(* IEC 61131-3 sources: SmartHomeNew/ (part 11) *)

(* ---- PRG_Config_Staged_Change_Monitor.st ---- *)
PROGRAM PRG_Config_Staged_Change_Monitor
// ==============================================================================
// CONFIG STAGED CHANGE MONITOR
// ==============================================================================
// Tracks generic staged config fields controlled by GVL_CONFIG_CONTROL. When any
// staged value changes, the staged config version is incremented so HMI validation
// cannot be reused for a different draft.
// ==============================================================================
VAR
    L_Initialized : BOOL;
    L_Changed : BOOL;

    L_Last_STG_Reputation_Learning_Rate : REAL;
    L_Last_STG_Reputation_Recovery_Decay : REAL;
    L_Last_STG_Min_Sensor_Confidence : REAL;
    L_Last_STG_Bad_Spike_Confidence : REAL;
    L_Last_STG_Default_Confidence : REAL;

    L_Last_STG_Night_Start_Hour : INT;
    L_Last_STG_Night_End_Hour : INT;
    L_Last_STG_VentBoost_Humidity_Threshold : REAL;

    L_Last_STG_Stabilization_Delay_MS : UDINT;

    L_Last_STG_PLC_Inactive_Close_Gas : BOOL;
    L_Last_STG_PLC_Inactive_Stop_Boiler : BOOL;
    L_Last_STG_PLC_Inactive_Block_Heating : BOOL;
    L_Last_STG_PLC_Inactive_Stop_Vent : BOOL;
    L_Last_STG_PLC_Inactive_Block_Water : BOOL;
END_VAR

L_Changed := FALSE;

IF NOT L_Initialized THEN
    L_Initialized := TRUE;
ELSE
    IF L_Last_STG_Reputation_Learning_Rate <> GVL_CONFIG_CONTROL.STG_Reputation_Learning_Rate THEN L_Changed := TRUE; END_IF;
    IF L_Last_STG_Reputation_Recovery_Decay <> GVL_CONFIG_CONTROL.STG_Reputation_Recovery_Decay THEN L_Changed := TRUE; END_IF;
    IF L_Last_STG_Min_Sensor_Confidence <> GVL_CONFIG_CONTROL.STG_Min_Sensor_Confidence THEN L_Changed := TRUE; END_IF;
    IF L_Last_STG_Bad_Spike_Confidence <> GVL_CONFIG_CONTROL.STG_Bad_Spike_Confidence THEN L_Changed := TRUE; END_IF;
    IF L_Last_STG_Default_Confidence <> GVL_CONFIG_CONTROL.STG_Default_Confidence THEN L_Changed := TRUE; END_IF;

    IF L_Last_STG_Night_Start_Hour <> GVL_CONFIG_CONTROL.STG_Night_Start_Hour THEN L_Changed := TRUE; END_IF;
    IF L_Last_STG_Night_End_Hour <> GVL_CONFIG_CONTROL.STG_Night_End_Hour THEN L_Changed := TRUE; END_IF;
    IF L_Last_STG_VentBoost_Humidity_Threshold <> GVL_CONFIG_CONTROL.STG_VentBoost_Humidity_Threshold THEN L_Changed := TRUE; END_IF;

    IF L_Last_STG_Stabilization_Delay_MS <> GVL_CONFIG_CONTROL.STG_Stabilization_Delay_MS THEN L_Changed := TRUE; END_IF;

    IF L_Last_STG_PLC_Inactive_Close_Gas <> GVL_CONFIG_CONTROL.STG_PLC_Inactive_Close_Gas THEN L_Changed := TRUE; END_IF;
    IF L_Last_STG_PLC_Inactive_Stop_Boiler <> GVL_CONFIG_CONTROL.STG_PLC_Inactive_Stop_Boiler THEN L_Changed := TRUE; END_IF;
    IF L_Last_STG_PLC_Inactive_Block_Heating <> GVL_CONFIG_CONTROL.STG_PLC_Inactive_Block_Heating THEN L_Changed := TRUE; END_IF;
    IF L_Last_STG_PLC_Inactive_Stop_Vent <> GVL_CONFIG_CONTROL.STG_PLC_Inactive_Stop_Vent THEN L_Changed := TRUE; END_IF;
    IF L_Last_STG_PLC_Inactive_Block_Water <> GVL_CONFIG_CONTROL.STG_PLC_Inactive_Block_Water THEN L_Changed := TRUE; END_IF;
END_IF;

IF L_Changed THEN
    GVL_CONFIG_CONTROL.G_Staged_Config_Version := GVL_CONFIG_CONTROL.G_Staged_Config_Version + 1;
    GVL_CONFIG_CONTROL.G_Staged_Last_Changed_MS := GVL_TIME_SERVICE.G_Now_MS;
END_IF;

L_Last_STG_Reputation_Learning_Rate := GVL_CONFIG_CONTROL.STG_Reputation_Learning_Rate;
L_Last_STG_Reputation_Recovery_Decay := GVL_CONFIG_CONTROL.STG_Reputation_Recovery_Decay;
L_Last_STG_Min_Sensor_Confidence := GVL_CONFIG_CONTROL.STG_Min_Sensor_Confidence;
L_Last_STG_Bad_Spike_Confidence := GVL_CONFIG_CONTROL.STG_Bad_Spike_Confidence;
L_Last_STG_Default_Confidence := GVL_CONFIG_CONTROL.STG_Default_Confidence;

L_Last_STG_Night_Start_Hour := GVL_CONFIG_CONTROL.STG_Night_Start_Hour;
L_Last_STG_Night_End_Hour := GVL_CONFIG_CONTROL.STG_Night_End_Hour;
L_Last_STG_VentBoost_Humidity_Threshold := GVL_CONFIG_CONTROL.STG_VentBoost_Humidity_Threshold;

L_Last_STG_Stabilization_Delay_MS := GVL_CONFIG_CONTROL.STG_Stabilization_Delay_MS;

L_Last_STG_PLC_Inactive_Close_Gas := GVL_CONFIG_CONTROL.STG_PLC_Inactive_Close_Gas;
L_Last_STG_PLC_Inactive_Stop_Boiler := GVL_CONFIG_CONTROL.STG_PLC_Inactive_Stop_Boiler;
L_Last_STG_PLC_Inactive_Block_Heating := GVL_CONFIG_CONTROL.STG_PLC_Inactive_Block_Heating;
L_Last_STG_PLC_Inactive_Stop_Vent := GVL_CONFIG_CONTROL.STG_PLC_Inactive_Stop_Vent;
L_Last_STG_PLC_Inactive_Block_Water := GVL_CONFIG_CONTROL.STG_PLC_Inactive_Block_Water;

// >>> BULK_SYNC_ANCHOR: PRG_Config_Staged_Change_Monitor <<<
END_PROGRAM

(* ---- PRG_Config_Validation.st ---- *)
PROGRAM PRG_Config_Validation
VAR
    fbConfigSimulation : FB_Config_Simulation;

    L_i : INT;
    L_Zone : INT;
    L_Sensor : INT;
    L_Manifold : INT;
    L_Map_Index : INT;
    L_Config_Error : BOOL;
END_VAR

// ======================================================
// CENTRAL CONFIGURATION VALIDATION
// ======================================================
// Diagnostic-only layer.
//
// This PRG may set validation/configuration status flags and text,
// but must not directly mutate aggregated diagnostics fields.
// Aggregated diagnostics ownership is centralized in:
//
//   FB_System_Health_Orchestrator
//
// This PRG also must not write command/shadow/output structures.
// ======================================================

L_Config_Error := FALSE;

// ======================================================
// ACTIVE SIZE CONFIGURATION
// ======================================================
IF (GVL_SYSTEM_SIZE_CONFIG.G_Active_Heating_Circuits < 1) OR
   (GVL_SYSTEM_SIZE_CONFIG.G_Active_Heating_Circuits > GVL_CONSTANTS.C_MAX_HEATING_CIRCUITS) THEN
    L_Config_Error := TRUE;
END_IF;

IF (GVL_SYSTEM_SIZE_CONFIG.G_Active_Water_Zones < 1) OR
   (GVL_SYSTEM_SIZE_CONFIG.G_Active_Water_Zones > GVL_CONSTANTS.C_MAX_WATER_ZONES) THEN
    L_Config_Error := TRUE;
END_IF;

IF (GVL_SYSTEM_SIZE_CONFIG.G_Active_Light_Zones < 1) OR
   (GVL_SYSTEM_SIZE_CONFIG.G_Active_Light_Zones > GVL_CONSTANTS.C_MAX_LIGHT_ZONES) THEN
    L_Config_Error := TRUE;
END_IF;

IF (GVL_SYSTEM_SIZE_CONFIG.G_Active_Blinds < 0) OR
   (GVL_SYSTEM_SIZE_CONFIG.G_Active_Blinds > GVL_CONSTANTS.C_MAX_BLINDS) THEN
    L_Config_Error := TRUE;
END_IF;

IF (GVL_SYSTEM_SIZE_CONFIG.G_Active_Sockets < 0) OR
   (GVL_SYSTEM_SIZE_CONFIG.G_Active_Sockets > GVL_CONSTANTS.C_MAX_SOCKETS) THEN
    L_Config_Error := TRUE;
END_IF;

// ======================================================
// HEATING CIRCUIT CONFIGURATION
// ======================================================
FOR L_i := 1 TO GVL_CONSTANTS.C_MAX_HEATING_CIRCUITS DO
    L_Zone := BYTE_TO_INT(GVL_CONFIG.G_HMI_FloorHeating_Configs[L_i].zone);
    L_Sensor := BYTE_TO_INT(GVL_CONFIG.G_HMI_FloorHeating_Configs[L_i].sensor_id);
    L_Manifold := BYTE_TO_INT(GVL_CONFIG.G_HMI_FloorHeating_Configs[L_i].manifold_id);

    IF (L_Zone < 1) OR (L_Zone > GVL_CONSTANTS.C_MAX_ZONES) THEN
        L_Config_Error := TRUE;
    END_IF;

    IF (L_Sensor < 1) OR (L_Sensor > GVL_CONSTANTS.C_MAX_ZONES) THEN
        L_Config_Error := TRUE;
    END_IF;

    IF (L_Manifold < 1) OR (L_Manifold > GVL_CONSTANTS.C_MAX_MANIFOLDS) THEN
        L_Config_Error := TRUE;
    END_IF;

    IF GVL_CONFIG.G_HMI_FloorHeating_Configs[L_i].min_temp > GVL_CONFIG.G_HMI_FloorHeating_Configs[L_i].max_temp THEN
        L_Config_Error := TRUE;
    END_IF;
END_FOR;

IF (GVL_CONFIG.G_Max_Active_Manifolds < 1) OR
   (GVL_CONFIG.G_Max_Active_Manifolds > GVL_CONSTANTS.C_MAX_MANIFOLDS) THEN
    L_Config_Error := TRUE;
END_IF;

IF GVL_CONFIG.G_Max_Thermal_Budget <= 0.0 THEN
    L_Config_Error := TRUE;
END_IF;

IF GVL_CONFIG.G_Policy_Min_Hold_MS < 10000 THEN
    L_Config_Error := TRUE;
END_IF;

// ======================================================
// ACCESS / TIMING CONFIGURATION
// ======================================================
IF (GVL_CONFIG.G_Access_Pulse_MS < 100) OR (GVL_CONFIG.G_Access_Pulse_MS > 5000) THEN
    L_Config_Error := TRUE;
END_IF;

// ======================================================
// MAP CONFIGURATION
// ======================================================
FOR L_i := 1 TO GVL_CONSTANTS.C_MAX_DOOR_SENSORS DO
    L_Map_Index := GVL_CONFIG.G_Door_Map[L_i];
    IF (L_Map_Index < 1) OR (L_Map_Index > GVL_CONSTANTS.C_MAX_SECURITY_SENSORS) THEN
        L_Config_Error := TRUE;
    END_IF;
END_FOR;

FOR L_i := 1 TO GVL_CONSTANTS.C_MAX_ZONES DO
    L_Map_Index := GVL_CONFIG.G_Window_Map[L_i];
    IF L_Map_Index <> 0 THEN
        IF (L_Map_Index < 1) OR (L_Map_Index > (GVL_CONSTANTS.C_MAX_SECURITY_SENSORS * 2)) THEN
            L_Config_Error := TRUE;
        END_IF;
    END_IF;
END_FOR;

FOR L_i := 1 TO GVL_CONSTANTS.C_MAX_HEATING_CIRCUITS DO
    IF (GVL_CONFIG.G_FloorTemp_Map[L_i] < 1) OR (GVL_CONFIG.G_FloorTemp_Map[L_i] > GVL_CONSTANTS.C_MAX_ZONES) THEN
        L_Config_Error := TRUE;
    END_IF;
END_FOR;

FOR L_i := 1 TO GVL_CONSTANTS.C_MAX_ZONES DO
    IF (GVL_CONFIG.G_RoomTemp_Map[L_i] < 1) OR (GVL_CONFIG.G_RoomTemp_Map[L_i] > GVL_CONSTANTS.C_MAX_ZONES) THEN
        L_Config_Error := TRUE;
    END_IF;
END_FOR;

// ======================================================
// HARDWARE SERVICE / RETRY CONFIGURATION
// ======================================================
IF GVL_CONFIG.G_Freeze_Hardware_Retry_Count < 0 THEN
    L_Config_Error := TRUE;
END_IF;

IF GVL_CONFIG.G_Freeze_Hardware_Retry_Delay_MS < 1000 THEN
    L_Config_Error := TRUE;
END_IF;

IF GVL_CONFIG.G_Pump_Exercise_Enabled THEN
    IF GVL_CONFIG.G_Pump_Exercise_Interval_MS < GVL_CONSTANTS.C_MS_IN_MINUTE THEN
        L_Config_Error := TRUE;
    END_IF;
    IF GVL_CONFIG.G_Pump_Exercise_Duration_MS < 1000 THEN
        L_Config_Error := TRUE;
    END_IF;
END_IF;

IF GVL_CONFIG.G_Water_Valve_Exercise_Enabled THEN
    IF GVL_CONFIG.G_Water_Valve_Exercise_Interval_MS < GVL_CONSTANTS.C_MS_IN_MINUTE THEN
        L_Config_Error := TRUE;
    END_IF;
    IF GVL_CONFIG.G_Water_Valve_Exercise_Duration_MS < 1000 THEN
        L_Config_Error := TRUE;
    END_IF;
END_IF;

IF GVL_CONFIG.G_Water_Valve_Close_Retry_Count < 0 THEN
    L_Config_Error := TRUE;
END_IF;

IF GVL_CONFIG.G_Water_Valve_Close_Retry_Delay_MS < 1000 THEN
    L_Config_Error := TRUE;
END_IF;

// ======================================================
// OPENTHERM / MODBUS RTU CONFIGURATION
// ======================================================
IF GVL_CONFIG.G_OpenTherm_Enabled THEN

    IF GVL_CONFIG.G_OpenTherm_Heartbeat_Timeout_MS < 1000 THEN
        L_Config_Error := TRUE;
    END_IF;

    IF GVL_CONFIG.G_OpenTherm_Command_Ack_Timeout_MS < 500 THEN
        L_Config_Error := TRUE;
    END_IF;

    IF GVL_CONFIG.G_Modbus_RTU_Baudrate < 1200 THEN
        L_Config_Error := TRUE;
    END_IF;

    IF (GVL_CONFIG.G_Modbus_RTU_Parity > 2) THEN
        L_Config_Error := TRUE;
    END_IF;

    IF (GVL_CONFIG.G_Modbus_RTU_Stop_Bits < 1) OR
       (GVL_CONFIG.G_Modbus_RTU_Stop_Bits > 2) THEN
        L_Config_Error := TRUE;
    END_IF;

    IF (GVL_CONFIG.G_Modbus_RTU_Data_Bits < 7) OR
       (GVL_CONFIG.G_Modbus_RTU_Data_Bits > 8) THEN
        L_Config_Error := TRUE;
    END_IF;

    IF GVL_CONFIG.G_Modbus_RTU_Slave_ID = 0 THEN
        L_Config_Error := TRUE;
    END_IF;

    IF GVL_CONFIG.G_Modbus_RTU_Poll_Interval_MS < 50 THEN
        L_Config_Error := TRUE;
    END_IF;

    IF GVL_CONFIG.G_Modbus_RTU_Request_Timeout_MS < 50 THEN
        L_Config_Error := TRUE;
    END_IF;

    IF GVL_CONFIG.G_Modbus_RTU_Retry_Count < 0 THEN
        L_Config_Error := TRUE;
    END_IF;

    FOR L_i := 1 TO GVL_CONSTANTS.C_MAX_BOILERS DO
        IF GVL_CONFIG.G_OpenTherm_Register_Map[L_i].Cmd_Enable_Offset = GVL_CONFIG.G_OpenTherm_Register_Map[L_i].Status_Word_Offset THEN
            L_Config_Error := TRUE;
        END_IF;

        IF GVL_CONFIG.G_OpenTherm_Register_Map[L_i].Cmd_Setpoint_x10_Offset = GVL_CONFIG.G_OpenTherm_Register_Map[L_i].Status_Word_Offset THEN
            L_Config_Error := TRUE;
        END_IF;
    END_FOR;
END_IF;

// ======================================================
// SENSOR COUNT SANITY
// ======================================================
IF GVL_CONSTANTS.C_MAX_METHANE_SENSORS < 2 THEN
    L_Config_Error := TRUE;
END_IF;

IF GVL_CONSTANTS.C_MAX_SMOKE_SENSORS < 6 THEN
    L_Config_Error := TRUE;
END_IF;

IF GVL_CONSTANTS.C_MAX_CO_SENSORS < 8 THEN
    L_Config_Error := TRUE;
END_IF;

IF GVL_CONSTANTS.C_MAX_FLOOD_SENSORS < 9 THEN
    L_Config_Error := TRUE;
END_IF;

// ======================================================
// CONFIG SIMULATION / COMMISSIONING VALIDATION
// ======================================================
fbConfigSimulation(
    VI_Enable := TRUE,
    VI_Request := GVL_CONFIG_SIMULATION.G_Simulation_Request,
    VI_Confirm := GVL_CONFIG_SIMULATION.G_Simulation_Confirm
);

IF fbConfigSimulation.VO_Executed AND NOT fbConfigSimulation.VO_Result_OK THEN
    L_Config_Error := TRUE;
END_IF;

// ======================================================
// STORE FLAGS
// ======================================================
GVL_CONFIG_VALIDATION.G_Config_Valid := NOT L_Config_Error;
GVL_CONFIG_VALIDATION.G_Config_Critical_Error := L_Config_Error;
GVL_CONFIG_VALIDATION.G_Config_Last_Update_MS := GVL_STATUS.G_System_Time_MS;

IF L_Config_Error THEN
    GVL_CONFIG_VALIDATION.G_Config_Active_Error_Text := 'CONFIG VALIDATION ERROR';
    GVL_STATUS.G_System_Mode_Text := 'CONFIG ERROR';
ELSE
    GVL_CONFIG_VALIDATION.G_Config_Active_Error_Text := '';
END_IF;

IF GVL_CONFIG_VALIDATION.G_Config_Active_Error_Text <> '' THEN
    GVL_CONFIG_VALIDATION.G_Config_Last_Error_Text := GVL_CONFIG_VALIDATION.G_Config_Active_Error_Text;
ELSIF GVL_CONFIG_VALIDATION.G_Config_Control_Error_Text <> '' THEN
    GVL_CONFIG_VALIDATION.G_Config_Last_Error_Text := GVL_CONFIG_VALIDATION.G_Config_Control_Error_Text;
ELSE
    GVL_CONFIG_VALIDATION.G_Config_Last_Error_Text := '';
END_IF;

END_PROGRAM

(* ---- PRG_Config_Versioning.st ---- *)
PROGRAM PRG_Config_Versioning
VAR
    L_i : INT;
    L_Config_Error : BOOL;
END_VAR

// Detect config error from validation layer.
// Calibration processor faults are surfaced through Sensor_Fault, so the
// configuration rollback snapshot must include calibration records too.
L_Config_Error := GVL_STATUS.G_Diagnostics.Sensor_Fault OR GVL_STATUS.G_Diagnostics.Subsystem_Degraded;

// --- Save snapshot when system is healthy ---
IF NOT L_Config_Error THEN
    FOR L_i := 1 TO GVL_CONSTANTS.C_MAX_HEATING_CIRCUITS DO
        GVL_CONFIG_BACKUP.G_Backup_FloorHeating_Configs[L_i] := GVL_CONFIG.G_HMI_FloorHeating_Configs[L_i];
    END_FOR;

    GVL_CONFIG_BACKUP.G_Backup_Max_Active_Manifolds := GVL_CONFIG.G_Max_Active_Manifolds;
    GVL_CONFIG_BACKUP.G_Backup_Max_Thermal_Budget := GVL_CONFIG.G_Max_Thermal_Budget;

    GVL_CONFIG_BACKUP.G_Backup_Calib_Outdoor_Temp := GVL_CONFIG.G_Calib_Outdoor_Temp;
    GVL_CONFIG_BACKUP.G_Backup_Calib_Ambient_Lux := GVL_CONFIG.G_Calib_Ambient_Lux;

    FOR L_i := 1 TO GVL_CONSTANTS.C_MAX_SUPPLY_TEMPS DO
        GVL_CONFIG_BACKUP.G_Backup_Calib_Supply_Temps[L_i] := GVL_CONFIG.G_Calib_Supply_Temps[L_i];
    END_FOR;

    FOR L_i := 1 TO GVL_CONSTANTS.C_MAX_ZONES DO
        GVL_CONFIG_BACKUP.G_Backup_Calib_Room_Temps[L_i] := GVL_CONFIG.G_Calib_Room_Temps[L_i];
        GVL_CONFIG_BACKUP.G_Backup_Calib_Floor_Temps[L_i] := GVL_CONFIG.G_Calib_Floor_Temps[L_i];
        GVL_CONFIG_BACKUP.G_Backup_Calib_CO2[L_i] := GVL_CONFIG.G_Calib_CO2[L_i];
        GVL_CONFIG_BACKUP.G_Backup_Calib_Humidity[L_i] := GVL_CONFIG.G_Calib_Humidity[L_i];
    END_FOR;

    FOR L_i := 1 TO GVL_CONSTANTS.C_MAX_MANIFOLDS DO
        GVL_CONFIG_BACKUP.G_Backup_Calib_Manifold_T_Supply[L_i] := GVL_CONFIG.G_Calib_Manifold_T_Supply[L_i];
        GVL_CONFIG_BACKUP.G_Backup_Calib_Manifold_T_Return[L_i] := GVL_CONFIG.G_Calib_Manifold_T_Return[L_i];
    END_FOR;

    FOR L_i := 1 TO GVL_CONSTANTS.C_MAX_METHANE_SENSORS DO
        GVL_CONFIG_BACKUP.G_Backup_Calib_Methane[L_i] := GVL_CONFIG.G_Calib_Methane[L_i];
    END_FOR;

    FOR L_i := 1 TO GVL_CONSTANTS.C_MAX_CO_SENSORS DO
        GVL_CONFIG_BACKUP.G_Backup_Calib_CO[L_i] := GVL_CONFIG.G_Calib_CO[L_i];
    END_FOR;

    GVL_CONFIG_BACKUP.G_Backup_Valid := TRUE;
END_IF;

// --- Rollback if config invalid ---
IF L_Config_Error THEN

    // Freeze system via command layer
    GVL_COMMAND_SHADOW.G_Heating_Block := TRUE;
    GVL_COMMAND_SHADOW.G_Boiler_Stop := TRUE;

    // Restore snapshot only if valid
    IF GVL_CONFIG_BACKUP.G_Backup_Valid THEN
        FOR L_i := 1 TO GVL_CONSTANTS.C_MAX_HEATING_CIRCUITS DO
            GVL_CONFIG.G_HMI_FloorHeating_Configs[L_i] := GVL_CONFIG_BACKUP.G_Backup_FloorHeating_Configs[L_i];
        END_FOR;

        GVL_CONFIG.G_Max_Active_Manifolds := GVL_CONFIG_BACKUP.G_Backup_Max_Active_Manifolds;
        GVL_CONFIG.G_Max_Thermal_Budget := GVL_CONFIG_BACKUP.G_Backup_Max_Thermal_Budget;

        GVL_CONFIG.G_Calib_Outdoor_Temp := GVL_CONFIG_BACKUP.G_Backup_Calib_Outdoor_Temp;
        GVL_CONFIG.G_Calib_Ambient_Lux := GVL_CONFIG_BACKUP.G_Backup_Calib_Ambient_Lux;

        FOR L_i := 1 TO GVL_CONSTANTS.C_MAX_SUPPLY_TEMPS DO
            GVL_CONFIG.G_Calib_Supply_Temps[L_i] := GVL_CONFIG_BACKUP.G_Backup_Calib_Supply_Temps[L_i];
        END_FOR;

        FOR L_i := 1 TO GVL_CONSTANTS.C_MAX_ZONES DO
            GVL_CONFIG.G_Calib_Room_Temps[L_i] := GVL_CONFIG_BACKUP.G_Backup_Calib_Room_Temps[L_i];
            GVL_CONFIG.G_Calib_Floor_Temps[L_i] := GVL_CONFIG_BACKUP.G_Backup_Calib_Floor_Temps[L_i];
            GVL_CONFIG.G_Calib_CO2[L_i] := GVL_CONFIG_BACKUP.G_Backup_Calib_CO2[L_i];
            GVL_CONFIG.G_Calib_Humidity[L_i] := GVL_CONFIG_BACKUP.G_Backup_Calib_Humidity[L_i];
        END_FOR;

        FOR L_i := 1 TO GVL_CONSTANTS.C_MAX_MANIFOLDS DO
            GVL_CONFIG.G_Calib_Manifold_T_Supply[L_i] := GVL_CONFIG_BACKUP.G_Backup_Calib_Manifold_T_Supply[L_i];
            GVL_CONFIG.G_Calib_Manifold_T_Return[L_i] := GVL_CONFIG_BACKUP.G_Backup_Calib_Manifold_T_Return[L_i];
        END_FOR;

        FOR L_i := 1 TO GVL_CONSTANTS.C_MAX_METHANE_SENSORS DO
            GVL_CONFIG.G_Calib_Methane[L_i] := GVL_CONFIG_BACKUP.G_Backup_Calib_Methane[L_i];
        END_FOR;

        FOR L_i := 1 TO GVL_CONSTANTS.C_MAX_CO_SENSORS DO
            GVL_CONFIG.G_Calib_CO[L_i] := GVL_CONFIG_BACKUP.G_Backup_Calib_CO[L_i];
        END_FOR;

        GVL_STATUS.G_System_Mode_Text := 'CONFIG ROLLBACK';
    ELSE
        GVL_STATUS.G_System_Mode_Text := 'CONFIG INVALID - NO BACKUP';
    END_IF;
END_IF;

END_PROGRAM
// >>> BULK_SYNC_ANCHOR: PRG_Config_Versioning <<<

(* ---- PRG_Convergence_Governor.st ---- *)
PROGRAM PRG_Convergence_Governor
VAR
    L_Now_MS : UDINT;
    L_Healthy : BOOL := TRUE;
    L_Error_Code : UDINT := 0;
    L_Error_Text : STRING(160) := '';
END_VAR

L_Now_MS := GVL_STATUS.G_System_Time_MS;
L_Healthy := TRUE;
L_Error_Code := 0;
L_Error_Text := '';

GVL_CONVERGENCE.Convergence_Runtime_Barrier_OK :=
    GVL_RUNTIME_EPOCH.Runtime_Runtime_Barrier_OK
    AND GVL_RUNTIME_EPOCH.Runtime_IO_Publication_Allowed;

GVL_CONVERGENCE.Convergence_Runtime_Snapshot_OK :=
    GVL_RUNTIME_SNAPSHOT.Snapshot_Frozen
    AND GVL_RUNTIME_SNAPSHOT.Snapshot_Publication_Allowed
    AND GVL_RUNTIME_SNAPSHOT.Snapshot_Copy_Valid
    AND GVL_RUNTIME_SNAPSHOT.Snapshot_Isolation_Valid
    AND GVL_RUNTIME_SNAPSHOT.Snapshot_Runtime_Authority_Valid
    AND NOT GVL_RUNTIME_SNAPSHOT.Snapshot_Mutation_Detected;

GVL_CONVERGENCE.Convergence_Distributed_Snapshot_OK :=
    GVL_DISTRIBUTED_SNAPSHOT.Distributed_Publication_Reconciled
    AND GVL_DISTRIBUTED_SNAPSHOT.Distributed_Publication_Freeze_Valid
    AND GVL_DISTRIBUTED_SNAPSHOT.Distributed_Snapshot_Consistent;

GVL_CONVERGENCE.Convergence_Distributed_Commit_OK :=
    GVL_DISTRIBUTED_COMMIT.Distributed_Commit_Valid
    AND GVL_DISTRIBUTED_COMMIT.Publication_Prepare_Valid
    AND GVL_DISTRIBUTED_COMMIT.Publication_Commit_Confirmed
    AND NOT GVL_DISTRIBUTED_COMMIT.Peer_Commit_Mismatch
    AND NOT GVL_DISTRIBUTED_COMMIT.Commit_Lease_Expired;

GVL_CONVERGENCE.Convergence_Semantic_Progress_OK :=
    GVL_SEMANTIC_PROGRESS.Semantic_Forward_Progress_Valid
    AND GVL_SEMANTIC_PROGRESS.Semantic_Execution_Continuity_OK
    AND NOT GVL_SEMANTIC_PROGRESS.Semantic_Stagnation_Detected
    AND NOT GVL_SEMANTIC_PROGRESS.Semantic_Replay_Suspected
    AND NOT GVL_SEMANTIC_PROGRESS.Semantic_Livelock_Suspected
    AND NOT GVL_SEMANTIC_PROGRESS.Semantic_Deadlock_Suspected
    AND NOT GVL_SEMANTIC_PROGRESS.Semantic_Progress_Lease_Expired
    AND NOT GVL_SEMANTIC_PROGRESS.Semantic_Progress_Quarantine_Active;

// Finalized output publication continuity.
GVL_CONVERGENCE.Convergence_Output_Freshness_OK :=
    GVL_RUNTIME_EPOCH.Runtime_Runtime_Barrier_OK
    AND GVL_RUNTIME_EPOCH.Runtime_IO_Publication_Allowed
    AND GVL_RUNTIME_SNAPSHOT.Snapshot_Frozen
    AND GVL_RUNTIME_SNAPSHOT.Snapshot_Publication_Allowed
    AND GVL_RUNTIME_SNAPSHOT.Snapshot_Copy_Valid
    AND GVL_RUNTIME_SNAPSHOT.Snapshot_Isolation_Valid
    AND NOT GVL_RUNTIME_SNAPSHOT.Snapshot_Mutation_Detected
    AND GVL_DISTRIBUTED_SNAPSHOT.Distributed_Publication_Reconciled
    AND GVL_DISTRIBUTED_SNAPSHOT.Distributed_Publication_Freeze_Valid
    AND GVL_DISTRIBUTED_SNAPSHOT.Distributed_Snapshot_Consistent
    AND GVL_DISTRIBUTED_COMMIT.Distributed_Commit_Valid
    AND GVL_DISTRIBUTED_COMMIT.Publication_Prepare_Valid
    AND GVL_DISTRIBUTED_COMMIT.Publication_Commit_Confirmed
    AND NOT GVL_DISTRIBUTED_COMMIT.Peer_Commit_Mismatch
    AND NOT GVL_DISTRIBUTED_COMMIT.Commit_Lease_Expired
    AND GVL_OUTPUT_EPOCH.Output_Publication_Valid
    AND GVL_OUTPUT_EPOCH.Output_Runtime_Epoch_Valid
    AND NOT GVL_OUTPUT_EPOCH.Output_Lease_Expired
    AND NOT GVL_OUTPUT_EPOCH.Output_Forced_Safe_Decay
    AND GVL_COMMAND_VERIFY.PreOutput_Barrier_OK
    AND NOT GVL_COMMAND_VERIFY.PreOutput_Block_IO;

IF NOT GVL_CONVERGENCE.Convergence_Runtime_Barrier_OK THEN
    L_Healthy := FALSE;
    L_Error_Code := 18000;
    L_Error_Text := 'Runtime barrier convergence invalid';
END_IF;

IF L_Healthy AND NOT GVL_CONVERGENCE.Convergence_Runtime_Snapshot_OK THEN
    L_Healthy := FALSE;
    L_Error_Code := 18001;
    L_Error_Text := 'Runtime snapshot convergence invalid';
END_IF;

IF L_Healthy AND NOT GVL_CONVERGENCE.Convergence_Distributed_Snapshot_OK THEN
    L_Healthy := FALSE;
    L_Error_Code := 18002;
    L_Error_Text := 'Distributed snapshot convergence invalid';
END_IF;

IF L_Healthy AND NOT GVL_CONVERGENCE.Convergence_Distributed_Commit_OK THEN
    L_Healthy := FALSE;
    L_Error_Code := 18003;
    L_Error_Text := 'Distributed commit convergence invalid';
END_IF;

IF L_Healthy AND NOT GVL_CONVERGENCE.Convergence_Semantic_Progress_OK THEN
    L_Healthy := FALSE;
    L_Error_Code := 18004;
    L_Error_Text := 'Semantic progress convergence invalid';
END_IF;

IF L_Healthy AND NOT GVL_CONVERGENCE.Convergence_Output_Freshness_OK THEN
    L_Healthy := FALSE;
    L_Error_Code := 18005;
    L_Error_Text := 'Output freshness convergence invalid';
END_IF;

IF L_Healthy THEN
    GVL_CONVERGENCE.Convergence_Healthy_Observed := TRUE;

    GVL_CONVERGENCE.Recovery_Stable_Cycle_Count :=
        GVL_CONVERGENCE.Recovery_Stable_Cycle_Count + 1;

    IF GVL_CONVERGENCE.Convergence_Last_Healthy_MS = 0 THEN
        GVL_CONVERGENCE.Convergence_Last_Healthy_MS := L_Now_MS;
    END_IF;

    GVL_CONVERGENCE.Recovery_Stable_Time_MS :=
        L_Now_MS - GVL_CONVERGENCE.Convergence_Last_Healthy_MS;

    IF (GVL_CONVERGENCE.Recovery_Stable_Cycle_Count >= GVL_CONVERGENCE.Convergence_Min_Stable_Cycles)
    AND (GVL_CONVERGENCE.Recovery_Stable_Time_MS >= GVL_CONVERGENCE.Convergence_Min_Stable_Time_MS) THEN
        GVL_CONVERGENCE.Convergence_Lease_OK := TRUE;
        GVL_CONVERGENCE.Convergence_Release_Allowed := TRUE;
    ELSE
        GVL_CONVERGENCE.Convergence_Lease_OK := FALSE;
        GVL_CONVERGENCE.Convergence_Release_Allowed := FALSE;
    END_IF;

    GVL_CONVERGENCE.Convergence_Last_Error_Code := 0;
    GVL_CONVERGENCE.Convergence_Last_Error_Text := '';
ELSE
    GVL_CONVERGENCE.Convergence_Healthy_Observed := FALSE;

    GVL_CONVERGENCE.Recovery_Stable_Cycle_Count := 0;
    GVL_CONVERGENCE.Recovery_Stable_Time_MS := 0;

    GVL_CONVERGENCE.Convergence_Lease_OK := FALSE;
    GVL_CONVERGENCE.Convergence_Release_Allowed := FALSE;

    GVL_CONVERGENCE.Convergence_Last_Healthy_MS := 0;
    GVL_CONVERGENCE.Convergence_Last_Invalidation_MS := L_Now_MS;

    GVL_CONVERGENCE.Convergence_Invalidation_Count :=
        GVL_CONVERGENCE.Convergence_Invalidation_Count + 1;

    GVL_CONVERGENCE.Convergence_Last_Error_Code := L_Error_Code;
    GVL_CONVERGENCE.Convergence_Last_Error_Text := L_Error_Text;
END_IF;

END_PROGRAM

(* ---- PRG_Debug_View.st ---- *)
PROGRAM PRG_Debug_View
VAR
    L_i : INT;
    L_MaxWeight : REAL;
    L_MinWeight : REAL;
    L_Weight : REAL;
    L_Index : INT;
END_VAR

GVL_DEBUG_VIEW.D_Current_Time_MS := GVL_TIME_SERVICE.G_Now_MS;

GVL_DEBUG_VIEW.D_Safety_Mode := GVL_SAFETY_SHUTDOWN.G_Safety_Mode;
GVL_DEBUG_VIEW.D_Safety_Active := (GVL_SAFETY_SHUTDOWN.G_Safety_Mode <> NORMAL);
GVL_DEBUG_VIEW.D_Recovery_Phase := GVL_SAFETY_RECOVERY.G_Recovery_Phase;
GVL_DEBUG_VIEW.D_Recovery_Active := GVL_SAFETY_RECOVERY.G_Recovery_Active;

GVL_DEBUG_VIEW.D_Current_Scenario := GVL_INTENT_BEHAVIOR.I_Selected_Scenario_Text;
GVL_DEBUG_VIEW.D_Behavior_Reason := GVL_INTENT_BEHAVIOR.I_Reason_Text;

GVL_DEBUG_VIEW.D_Score_Night := GVL_INTENT_BEHAVIOR.I_Score_Night;
GVL_DEBUG_VIEW.D_Score_Preheat := GVL_INTENT_BEHAVIOR.I_Score_Preheat;
GVL_DEBUG_VIEW.D_Score_VentBoost := GVL_INTENT_BEHAVIOR.I_Score_Vent_Boost;
GVL_DEBUG_VIEW.D_Score_AccessSecure := GVL_INTENT_BEHAVIOR.I_Score_Access_Secure;

GVL_DEBUG_VIEW.D_Intent_Night := GVL_INTENT_BEHAVIOR.I_Request_Night_Mode;
GVL_DEBUG_VIEW.D_Intent_Comfort := GVL_INTENT_BEHAVIOR.I_Request_Comfort_Mode;
GVL_DEBUG_VIEW.D_Intent_VentBoost := GVL_INTENT_BEHAVIOR.I_Request_Ventilation_Boost;
GVL_DEBUG_VIEW.D_Intent_AccessSecure := GVL_INTENT_BEHAVIOR.I_Request_Access_Secure_Mode;

GVL_DEBUG_VIEW.D_Heating_Block := GVL_COMMAND_SHADOW.G_Heating_Block;
GVL_DEBUG_VIEW.D_Vent_Stop := GVL_COMMAND_SHADOW.G_Vent_Stop;
GVL_DEBUG_VIEW.D_Water_Block := GVL_COMMAND_SHADOW.G_Water_Block;
GVL_DEBUG_VIEW.D_Access_Open_Active := GVL_COMMAND_SHADOW.G_Gate_Open OR GVL_COMMAND_SHADOW.G_Wicket_Open;

GVL_DEBUG_VIEW.D_Global_Reason := GVL_EXPLAINABILITY.G_Last_Global_Reason_Text;
GVL_DEBUG_VIEW.D_Behavior_Why_Active := GVL_EXPLAINABILITY.G_Behavior_Why_Active;
GVL_DEBUG_VIEW.D_Heating_Why_Blocked := GVL_EXPLAINABILITY.G_Heating_Why_Blocked;
GVL_DEBUG_VIEW.D_Vent_Why_Stopped := GVL_EXPLAINABILITY.G_Vent_Why_Stopped;
GVL_DEBUG_VIEW.D_Water_Why_Closed := GVL_EXPLAINABILITY.G_Water_Why_Closed;
GVL_DEBUG_VIEW.D_Access_Why_Opened := GVL_EXPLAINABILITY.G_Access_Why_Opened;

// MAIN PHASE FEEDBACK SUMMARY -> DEBUG VIEW
GVL_DEBUG_VIEW.D_Main_Phase_Current := GVL_MAIN_PHASE_FEEDBACK.G_Current_Phase;
GVL_DEBUG_VIEW.D_Main_Phase_Critical_Executed := GVL_MAIN_PHASE_FEEDBACK.G_Critical_Path_Executed;
GVL_DEBUG_VIEW.D_Main_Phase_Critical_Valid := GVL_MAIN_PHASE_FEEDBACK.G_Critical_Path_Valid;
GVL_DEBUG_VIEW.D_Main_Phase_Observability_Executed := GVL_MAIN_PHASE_FEEDBACK.G_Observability_Path_Executed;
GVL_DEBUG_VIEW.D_Main_Phase_Observability_Valid := GVL_MAIN_PHASE_FEEDBACK.G_Observability_Path_Valid;
GVL_DEBUG_VIEW.D_Main_Phase_Any_Invalid := GVL_MAIN_PHASE_FEEDBACK.G_Any_Phase_Invalid;
GVL_DEBUG_VIEW.D_Main_Phase_Status_Code := GVL_MAIN_PHASE_FEEDBACK.G_Status_Code;
GVL_DEBUG_VIEW.D_Main_Phase_Status_Text := GVL_MAIN_PHASE_FEEDBACK.G_Status_Text;

// SENSOR QUALITY → HMI
GVL_DEBUG_VIEW.D_Input_Source_Valid := GVL_INPUT.IN_Source_Valid;
GVL_DEBUG_VIEW.D_Input_Degraded := GVL_INPUT.IN_Input_Degraded;
GVL_DEBUG_VIEW.D_Sensor_Fault := GVL_INPUT.IN_Sensor_Fault;
GVL_DEBUG_VIEW.D_Validation_Failed := GVL_INPUT.IN_Validation_Failed;
GVL_DEBUG_VIEW.D_Anomaly_Detected := GVL_INPUT.IN_Anomaly_Detected;
GVL_DEBUG_VIEW.D_Validation_Reason := GVL_INPUT.IN_Validation_Reason;
GVL_DEBUG_VIEW.D_Anomaly_Reason := GVL_INPUT.IN_Anomaly_Reason;
GVL_DEBUG_VIEW.D_Last_Invalid_Zone := GVL_INPUT.IN_Last_Invalid_Zone;
GVL_DEBUG_VIEW.D_Min_Zone_Confidence := GVL_INPUT.IN_Min_Zone_Confidence;
GVL_DEBUG_VIEW.D_Worst_Zone := GVL_INPUT.IN_Worst_Zone;

GVL_DEBUG_VIEW.D_Adapt_Profile := GVL_BEHAVIOR_ADAPT.G_Adapt_Profile;

IF GVL_BEHAVIOR_ADAPT.G_Adapt_Profile = ADAPT_PROFILE_STABLE THEN
    GVL_DEBUG_VIEW.D_Adapt_Profile_Text := 'STABLE';
ELSIF GVL_BEHAVIOR_ADAPT.G_Adapt_Profile = ADAPT_PROFILE_BALANCED THEN
    GVL_DEBUG_VIEW.D_Adapt_Profile_Text := 'BALANCED';
ELSE
    GVL_DEBUG_VIEW.D_Adapt_Profile_Text := 'AGGRESSIVE';
END_IF;

L_MaxWeight := 0.0;
L_MinWeight := 9999.0;
GVL_DEBUG_VIEW.D_Main_VentBoost_Zone := 0;

FOR L_i := 1 TO GVL_CONSTANTS.C_MAX_ZONES DO
    L_Weight := GVL_BEHAVIOR_ADAPT.G_VentBoost_Zone_Adapt[L_i].Zone_Weight;
    IF L_Weight > L_MaxWeight THEN
        L_MaxWeight := L_Weight;
        GVL_DEBUG_VIEW.D_Main_VentBoost_Zone := L_i;
        GVL_DEBUG_VIEW.D_Main_VentBoost_Zone_Weight := L_Weight;
        GVL_DEBUG_VIEW.D_Main_VentBoost_Zone_Confidence :=
            GVL_BEHAVIOR_ADAPT.G_VentBoost_Zone_Adapt[L_i].Confidence;
    END_IF;
    IF L_Weight < L_MinWeight THEN
        L_MinWeight := L_Weight;
    END_IF;
END_FOR;

GVL_DEBUG_VIEW.D_Max_VentBoost_Zone_Weight := L_MaxWeight;
GVL_DEBUG_VIEW.D_Min_VentBoost_Zone_Weight := L_MinWeight;

L_Index := GVL_TRACE.G_Trace_Write_Index - 1;
IF L_Index < 1 THEN
    L_Index := 200;
END_IF;

GVL_DEBUG_VIEW.D_Last_Trace_Text := GVL_TRACE.G_Trace_Buffer[L_Index].Text;
GVL_DEBUG_VIEW.D_Last_Trace_Time_MS := GVL_TRACE.G_Trace_Buffer[L_Index].Timestamp_MS;
GVL_DEBUG_VIEW.D_Last_Trace_Reason := GVL_TRACE.G_Trace_Buffer[L_Index].Reason_Code;

END_PROGRAM

(* ---- PRG_Deterministic_Recovery_Path_Governor.st ---- *)
PROGRAM PRG_Deterministic_Recovery_Path_Governor
VAR
    L_Now_MS : UDINT;
END_VAR

L_Now_MS := GVL_STATUS.G_System_Time_MS;

IF GVL_CROSSDOMAIN_FAILSAFE_CLOSURE_FABRIC.CrossDomain_FailSafe_Closure_Granted
AND NOT GVL_DETERMINISTIC_RECOVERY_PATH_FABRIC.Unsafe_Recovery_Path_Detected
AND NOT GVL_DETERMINISTIC_RECOVERY_PATH_FABRIC.Recovery_Path_Divergence_Detected
AND NOT GVL_DETERMINISTIC_RECOVERY_PATH_FABRIC.Recovery_Causality_Break_Detected
AND NOT GVL_DETERMINISTIC_RECOVERY_PATH_FABRIC.Distributed_Recovery_Fork_Detected THEN

    GVL_DETERMINISTIC_RECOVERY_PATH_FABRIC.Deterministic_Recovery_Path_Valid := TRUE;
    GVL_DETERMINISTIC_RECOVERY_PATH_FABRIC.Deterministic_Recovery_Path_Granted := TRUE;
    GVL_DETERMINISTIC_RECOVERY_PATH_FABRIC.Deterministic_Recovery_Path_Canonical := TRUE;
    GVL_DETERMINISTIC_RECOVERY_PATH_FABRIC.Recovery_Lineage_Causality_Valid := TRUE;
    GVL_DETERMINISTIC_RECOVERY_PATH_FABRIC.Recovery_Physical_Convergence_Stable := TRUE;
    GVL_DETERMINISTIC_RECOVERY_PATH_FABRIC.Recovery_Timeline_Monotonic := TRUE;

    GVL_DETERMINISTIC_RECOVERY_PATH_FABRIC.Deterministic_Recovery_Path_Epoch :=
        GVL_CROSSDOMAIN_FAILSAFE_CLOSURE_FABRIC.CrossDomain_FailSafe_Closure_Epoch;

    GVL_DETERMINISTIC_RECOVERY_PATH_FABRIC.Deterministic_Recovery_Path_Last_Update_MS :=
        L_Now_MS;
END_IF;

END_PROGRAM

(* ---- PRG_Distributed_Commit_Governor.st ---- *)
PROGRAM PRG_Distributed_Commit_Governor
VAR
    L_Now_MS : UDINT;
    L_Delta_MS : UDINT;
    L_Commit_Valid : BOOL := TRUE;
    L_Error_Code : UDINT := 0;
    L_Error_Text : STRING(160) := '';
    L_Peer_Session_Active : BOOL := FALSE;

    L_Publication_Authority_Allowed : BOOL;
END_VAR

L_Now_MS := GVL_STATUS.G_System_Time_MS;
L_Commit_Valid := TRUE;
L_Error_Code := 0;
L_Error_Text := '';

// ======================================================
// DISTRIBUTED PUBLICATION COMMIT GOVERNOR
// ======================================================
// Governs deterministic peer publication commit continuity.
// Publication-authoritative only.
// Does not invalidate runtime barrier,
// PLC fencing or immutable snapshot authority.
//
// Recovery/release is convergence-lease based:
// distributed commit quarantine is not released on a
// single healthy scan.
//
// Distributed execution/publication authority is upstream.
// Observer-only nodes must never:
//   - participate in publication commit ownership;
//   - confirm publication authority;
//   - reopen publication continuity.
// ======================================================

GVL_DISTRIBUTED_COMMIT.Peer_Commit_Ack_Expired := FALSE;
GVL_DISTRIBUTED_COMMIT.Peer_Commit_Mismatch := FALSE;
GVL_DISTRIBUTED_COMMIT.Peer_Commit_Replay_Detected := FALSE;
GVL_DISTRIBUTED_COMMIT.Peer_Commit_Missing := FALSE;
GVL_DISTRIBUTED_COMMIT.Commit_Lease_Expired := FALSE;

L_Publication_Authority_Allowed :=
    GVL_Distributed_Execution_Gates.G_Runtime_Valid
    AND GVL_Distributed_Execution_Gates.G_Can_Replicate
    AND GVL_Distributed_Execution_Gates.G_Can_Own_Projection;

// ------------------------------------------------------
// Local publication projection.
// ------------------------------------------------------
// Distributed commit is upstream of output freshness in MAIN.
// Therefore local commit baseline must not read GVL_OUTPUT_EPOCH.
// It uses the already-prepared distributed snapshot epoch instead.
// ------------------------------------------------------

GVL_DISTRIBUTED_COMMIT.Local_Publication_Commit_Epoch := GVL_DISTRIBUTED_SNAPSHOT.Distributed_Snapshot_Epoch;
GVL_DISTRIBUTED_COMMIT.Local_Prepare_Epoch := GVL_DISTRIBUTED_SNAPSHOT.Distributed_Snapshot_Epoch;

// ------------------------------------------------------
// Distributed execution/publication authority.
// ------------------------------------------------------

IF NOT L_Publication_Authority_Allowed THEN

    L_Commit_Valid := FALSE;

    L_Error_Code := 14999;
    L_Error_Text :=
        'Distributed publication authority restricted';

END_IF;

// ------------------------------------------------------
// Immutable publication preparation validation.
// ------------------------------------------------------

IF L_Commit_Valid THEN

    IF GVL_DISTRIBUTED_SNAPSHOT.Distributed_Publication_Reconciled
    AND GVL_DISTRIBUTED_SNAPSHOT.Distributed_Publication_Freeze_Valid
    AND GVL_DISTRIBUTED_SNAPSHOT.Distributed_Snapshot_Consistent
    THEN
        GVL_DISTRIBUTED_COMMIT.Publication_Prepare_Active := TRUE;
        GVL_DISTRIBUTED_COMMIT.Publication_Prepare_Valid := TRUE;
    ELSE
        GVL_DISTRIBUTED_COMMIT.Publication_Prepare_Active := FALSE;
        GVL_DISTRIBUTED_COMMIT.Publication_Prepare_Valid := FALSE;

        L_Commit_Valid := FALSE;
        L_Error_Code := 15000;
        L_Error_Text := 'Distributed immutable publication prepare invalid';
    END_IF;

END_IF;

// ------------------------------------------------------
// Peer session detection.
// ------------------------------------------------------

IF GVL_DISTRIBUTED_COMMIT.Peer_Publication_Commit_Epoch > 0 THEN
    L_Peer_Session_Active := TRUE;
END_IF;

IF GVL_DISTRIBUTED_COMMIT.Peer_Prepare_Epoch > 0 THEN
    L_Peer_Session_Active := TRUE;
END_IF;

IF GVL_DISTRIBUTED_COMMIT.Peer_Commit_Ack_Valid THEN
    L_Peer_Session_Active := TRUE;
END_IF;

// ------------------------------------------------------
// Commit lease freshness validation.
// ------------------------------------------------------

IF L_Commit_Valid AND L_Peer_Session_Active THEN
    L_Delta_MS := L_Now_MS - GVL_DISTRIBUTED_COMMIT.Peer_Commit_Last_Refresh_MS;

    IF GVL_DISTRIBUTED_COMMIT.Commit_Lease_Active THEN
        IF L_Delta_MS > GVL_DISTRIBUTED_COMMIT.Commit_Timeout_MS THEN
            GVL_DISTRIBUTED_COMMIT.Commit_Lease_Expired := TRUE;

            L_Commit_Valid := FALSE;
            L_Error_Code := 15001;
            L_Error_Text := 'Distributed commit lease expired';
        END_IF;
    END_IF;
END_IF;

// ------------------------------------------------------
// Peer commit acknowledgement validation.
// ------------------------------------------------------

IF L_Commit_Valid AND L_Peer_Session_Active THEN
    IF NOT GVL_DISTRIBUTED_COMMIT.Peer_Commit_Ack_Valid THEN
        GVL_DISTRIBUTED_COMMIT.Peer_Commit_Missing := TRUE;

        L_Commit_Valid := FALSE;
        L_Error_Code := 15002;
        L_Error_Text := 'Peer commit acknowledgement missing';
    END_IF;
END_IF;

// ------------------------------------------------------
// Deterministic commit epoch continuity.
// ------------------------------------------------------

IF L_Commit_Valid AND L_Peer_Session_Active THEN
    IF GVL_DISTRIBUTED_COMMIT.Peer_Publication_Commit_Epoch < GVL_DISTRIBUTED_COMMIT.Local_Publication_Commit_Epoch THEN
        GVL_DISTRIBUTED_COMMIT.Peer_Commit_Mismatch := TRUE;

        L_Commit_Valid := FALSE;
        L_Error_Code := 15003;
        L_Error_Text := 'Peer commit epoch mismatch';
    END_IF;
END_IF;

// ------------------------------------------------------
// Replay protection foundation.
// ------------------------------------------------------

IF L_Commit_Valid AND L_Peer_Session_Active THEN
    IF GVL_DISTRIBUTED_COMMIT.Peer_Prepare_Epoch < GVL_DISTRIBUTED_COMMIT.Local_Prepare_Epoch THEN
        GVL_DISTRIBUTED_COMMIT.Peer_Commit_Replay_Detected := TRUE;

        L_Commit_Valid := FALSE;
        L_Error_Code := 15004;
        L_Error_Text := 'Peer commit replay detected';
    END_IF;
END_IF;

// ------------------------------------------------------
// Publish deterministic distributed commit state.
// ------------------------------------------------------

IF L_Commit_Valid THEN
    GVL_DISTRIBUTED_COMMIT.Distributed_Commit_Epoch := GVL_DISTRIBUTED_COMMIT.Distributed_Commit_Epoch + 1;
    GVL_DISTRIBUTED_COMMIT.Distributed_Commit_Reconciliation_Epoch := GVL_DISTRIBUTED_COMMIT.Distributed_Commit_Reconciliation_Epoch + 1;

    GVL_DISTRIBUTED_COMMIT.Publication_Commit_Requested := TRUE;

    IF L_Peer_Session_Active THEN
        GVL_DISTRIBUTED_COMMIT.Publication_Commit_Confirmed := TRUE;
        GVL_DISTRIBUTED_COMMIT.Commit_Lease_Active := TRUE;
    ELSE
        GVL_DISTRIBUTED_COMMIT.Publication_Commit_Confirmed := FALSE;
        GVL_DISTRIBUTED_COMMIT.Commit_Lease_Active := FALSE;
    END_IF;

    GVL_DISTRIBUTED_COMMIT.Distributed_Commit_Valid := TRUE;

    // Lease-based recovery release.
    IF GVL_CONVERGENCE.Convergence_Release_Allowed THEN
        GVL_DISTRIBUTED_COMMIT.Distributed_Commit_Quarantine_Active := FALSE;
    END_IF;

    GVL_DISTRIBUTED_COMMIT.Commit_Last_Reconciliation_MS := L_Now_MS;

    GVL_DISTRIBUTED_COMMIT.Distributed_Commit_Last_Error_Code := 0;
    GVL_DISTRIBUTED_COMMIT.Distributed_Commit_Last_Error_Text := '';
ELSE
    // Invalid distributed commit state escalates immediately.
    GVL_DISTRIBUTED_COMMIT.Publication_Commit_Confirmed := FALSE;

    GVL_DISTRIBUTED_COMMIT.Distributed_Commit_Valid := FALSE;
    GVL_DISTRIBUTED_COMMIT.Distributed_Commit_Quarantine_Active := TRUE;

    GVL_DISTRIBUTED_COMMIT.Distributed_Commit_Last_Error_Code := L_Error_Code;
    GVL_DISTRIBUTED_COMMIT.Distributed_Commit_Last_Error_Text := L_Error_Text;
END_IF;
END_PROGRAM

(* ---- PRG_Distributed_Commit_Ingestion.st ---- *)
PROGRAM PRG_Distributed_Commit_Ingestion
// ======================================================
// DISTRIBUTED COMMIT INGESTION
// ======================================================
// Explicit peer distributed commit ingestion layer.
//
// Purpose:
// normalize replicated peer commit-handshake state into
// distributed commit peer-input fields.
//
// This layer does NOT:
// - perform commit reconciliation
// - validate replay continuity
// - validate peer acknowledgements
// ======================================================

IF GVL_HA_SESSION_REPLICATION.HA_Remote_Session_Valid THEN
    GVL_DISTRIBUTED_COMMIT.Peer_Publication_Commit_Epoch :=
        GVL_HA_SESSION_REPLICATION.HA_Remote_Publication_Commit_Epoch;

    GVL_DISTRIBUTED_COMMIT.Peer_Prepare_Epoch :=
        GVL_HA_SESSION_REPLICATION.HA_Remote_Prepare_Epoch;

    GVL_DISTRIBUTED_COMMIT.Peer_Commit_Ack_Valid :=
        GVL_HA_SESSION_REPLICATION.HA_Remote_Commit_Ack_Valid;

    GVL_DISTRIBUTED_COMMIT.Peer_Commit_Last_Refresh_MS :=
        GVL_HA_SESSION_REPLICATION.HA_Remote_Commit_Last_Refresh_MS;
ELSE
    GVL_DISTRIBUTED_COMMIT.Peer_Publication_Commit_Epoch := 0;
    GVL_DISTRIBUTED_COMMIT.Peer_Prepare_Epoch := 0;
    GVL_DISTRIBUTED_COMMIT.Peer_Commit_Ack_Valid := FALSE;
    GVL_DISTRIBUTED_COMMIT.Peer_Commit_Last_Refresh_MS := 0;
END_IF;

// >>> BULK_SYNC_ANCHOR: PRG_Distributed_Commit_Ingestion <<<
END_PROGRAM

(* ---- PRG_Distributed_Commit_Observability.st ---- *)
PROGRAM PRG_Distributed_Commit_Observability
VAR
    L_Visibility_Required : BOOL := FALSE;
END_VAR

// ======================================================
// DISTRIBUTED COMMIT OBSERVABILITY GOVERNOR
// ======================================================
// Isolated downstream observability projection layer.
// Publication visibility only.
// Does not invalidate runtime barrier,
// PLC fencing, immutable snapshots or IO directly.
// ======================================================

GVL_OBSERVABILITY_AUTHORITY.Distributed_Commit_Visible := FALSE;
GVL_OBSERVABILITY_AUTHORITY.Distributed_Commit_Quarantine_Visible := FALSE;

GVL_OBSERVABILITY_AUTHORITY.Publication_Prepare_Visible := FALSE;
GVL_OBSERVABILITY_AUTHORITY.Publication_Commit_Visible := FALSE;

GVL_OBSERVABILITY_AUTHORITY.Peer_Commit_Ack_Visible := FALSE;
GVL_OBSERVABILITY_AUTHORITY.Peer_Commit_Mismatch_Visible := FALSE;
GVL_OBSERVABILITY_AUTHORITY.Peer_Commit_Replay_Visible := FALSE;
GVL_OBSERVABILITY_AUTHORITY.Peer_Commit_Missing_Visible := FALSE;

GVL_OBSERVABILITY_AUTHORITY.Commit_Lease_Expired_Visible := FALSE;

L_Visibility_Required := FALSE;

// ------------------------------------------------------
// Distributed commit validity visibility.
// ------------------------------------------------------

IF NOT GVL_DISTRIBUTED_COMMIT.Distributed_Commit_Valid THEN
    GVL_OBSERVABILITY_AUTHORITY.Distributed_Commit_Visible := TRUE;
    L_Visibility_Required := TRUE;
END_IF;

IF GVL_DISTRIBUTED_COMMIT.Distributed_Commit_Quarantine_Active THEN
    GVL_OBSERVABILITY_AUTHORITY.Distributed_Commit_Quarantine_Visible := TRUE;
    L_Visibility_Required := TRUE;
END_IF;

// ------------------------------------------------------
// Publication lifecycle visibility.
// ------------------------------------------------------

IF GVL_DISTRIBUTED_COMMIT.Publication_Prepare_Active THEN
    GVL_OBSERVABILITY_AUTHORITY.Publication_Prepare_Visible := TRUE;
END_IF;

IF GVL_DISTRIBUTED_COMMIT.Publication_Commit_Confirmed THEN
    GVL_OBSERVABILITY_AUTHORITY.Publication_Commit_Visible := TRUE;
END_IF;

// ------------------------------------------------------
// Peer commit continuity visibility.
// ------------------------------------------------------

IF GVL_DISTRIBUTED_COMMIT.Peer_Commit_Ack_Valid THEN
    GVL_OBSERVABILITY_AUTHORITY.Peer_Commit_Ack_Visible := TRUE;
END_IF;

IF GVL_DISTRIBUTED_COMMIT.Peer_Commit_Mismatch THEN
    GVL_OBSERVABILITY_AUTHORITY.Peer_Commit_Mismatch_Visible := TRUE;
    L_Visibility_Required := TRUE;
END_IF;

IF GVL_DISTRIBUTED_COMMIT.Peer_Commit_Replay_Detected THEN
    GVL_OBSERVABILITY_AUTHORITY.Peer_Commit_Replay_Visible := TRUE;
    L_Visibility_Required := TRUE;
END_IF;

IF GVL_DISTRIBUTED_COMMIT.Peer_Commit_Missing THEN
    GVL_OBSERVABILITY_AUTHORITY.Peer_Commit_Missing_Visible := TRUE;
    L_Visibility_Required := TRUE;
END_IF;

IF GVL_DISTRIBUTED_COMMIT.Commit_Lease_Expired THEN
    GVL_OBSERVABILITY_AUTHORITY.Commit_Lease_Expired_Visible := TRUE;
    L_Visibility_Required := TRUE;
END_IF;

// ------------------------------------------------------
// Downstream-only observability escalation.
// ------------------------------------------------------

IF L_Visibility_Required THEN
    GVL_OBSERVABILITY_AUTHORITY.Emergency_Visibility_Required := TRUE;
    GVL_OBSERVABILITY_AUTHORITY.Unsafe_State_Published := TRUE;
END_IF;
END_PROGRAM

(* ---- PRG_Distributed_Commit_Publication.st ---- *)
PROGRAM PRG_Distributed_Commit_Publication
// ======================================================
// DISTRIBUTED COMMIT PUBLICATION
// ======================================================
// Canonical local distributed commit export into the
// HA replication boundary.
//
// Purpose:
// publish normalized deterministic commit handshake state
// into the dedicated HA boundary before commit ingestion.
//
// This layer does NOT:
// - perform reconciliation
// - validate peer acknowledgements
// - arbitrate publication authority
//
// Disabled HA replication must not leave stale commit mirrors.
// ======================================================

IF NOT GVL_HA_SESSION_REPLICATION.HA_Replication_Enabled THEN
    GVL_HA_SESSION_REPLICATION.HA_Remote_Publication_Commit_Epoch := 0;
    GVL_HA_SESSION_REPLICATION.HA_Remote_Prepare_Epoch := 0;
    GVL_HA_SESSION_REPLICATION.HA_Remote_Commit_Ack_Valid := FALSE;
    GVL_HA_SESSION_REPLICATION.HA_Remote_Commit_Last_Refresh_MS := 0;
    RETURN;
END_IF;

GVL_HA_SESSION_REPLICATION.HA_Remote_Publication_Commit_Epoch :=
    GVL_DISTRIBUTED_COMMIT.Local_Publication_Commit_Epoch;

GVL_HA_SESSION_REPLICATION.HA_Remote_Prepare_Epoch :=
    GVL_DISTRIBUTED_COMMIT.Local_Prepare_Epoch;

GVL_HA_SESSION_REPLICATION.HA_Remote_Commit_Ack_Valid :=
    GVL_DISTRIBUTED_COMMIT.Publication_Commit_Confirmed;

GVL_HA_SESSION_REPLICATION.HA_Remote_Commit_Last_Refresh_MS :=
    GVL_STATUS.G_System_Time_MS;

// >>> BULK_SYNC_ANCHOR: PRG_Distributed_Commit_Publication <<<
END_PROGRAM

(* ---- PRG_Distributed_Epoch_Governor.st ---- *)
PROGRAM PRG_Distributed_Epoch_Governor
VAR
    L_Now_MS : UDINT;
    L_Delta_MS : UDINT;
    L_Distributed_Valid : BOOL := TRUE;
    L_Error_Code : UDINT := 0;
    L_Error_Text : STRING(160) := '';
    L_Peer_Session_Active : BOOL := FALSE;
END_VAR

L_Now_MS := GVL_STATUS.G_System_Time_MS;
L_Distributed_Valid := TRUE;
L_Error_Code := 0;
L_Error_Text := '';

// ======================================================
// DISTRIBUTED EPOCH GOVERNOR
// ======================================================
// Governs peer epoch reconciliation foundation.
// Prevents distributed stale authority continuity.
//
// Current implementation mode:
// peer-optional foundation mode.
//
// Missing peer topology is NOT treated as divergence.
// Peer validation activates only after real peer
// synchronization state exists.
// ======================================================

GVL_DISTRIBUTED_EPOCH.Peer_Lease_Expired := FALSE;
GVL_DISTRIBUTED_EPOCH.Peer_Snapshot_Stale := FALSE;
GVL_DISTRIBUTED_EPOCH.Peer_Runtime_Stale := FALSE;
GVL_DISTRIBUTED_EPOCH.Peer_Boot_Mismatch := FALSE;
GVL_DISTRIBUTED_EPOCH.Peer_Fencing_Conflict := FALSE;
GVL_DISTRIBUTED_EPOCH.Peer_Semantic_Continuity_Lost := FALSE;

// ------------------------------------------------------
// Local authority projection.
// ------------------------------------------------------

GVL_DISTRIBUTED_EPOCH.Local_Runtime_Epoch := GVL_RUNTIME_EPOCH.Runtime_Epoch;
GVL_DISTRIBUTED_EPOCH.Local_Snapshot_Epoch := GVL_RUNTIME_SNAPSHOT.Snapshot_Epoch;
GVL_DISTRIBUTED_EPOCH.Local_Boot_Generation := GVL_TIME_MONOTONIC.Boot_Generation_ID;
GVL_DISTRIBUTED_EPOCH.Local_Fencing_Token := GVL_PLC_FENCING.PLC_Fencing_Token;

// ------------------------------------------------------
// Peer session detection.
// ------------------------------------------------------
// Peer validation becomes authoritative only after
// real peer epoch continuity exists.
// ------------------------------------------------------

IF GVL_DISTRIBUTED_EPOCH.Peer_Runtime_Epoch > 0 THEN
    L_Peer_Session_Active := TRUE;
END_IF;

IF GVL_DISTRIBUTED_EPOCH.Peer_Snapshot_Epoch > 0 THEN
    L_Peer_Session_Active := TRUE;
END_IF;

IF GVL_DISTRIBUTED_EPOCH.Peer_Boot_Generation > 0 THEN
    L_Peer_Session_Active := TRUE;
END_IF;

IF GVL_DISTRIBUTED_EPOCH.Peer_Fencing_Token > 0 THEN
    L_Peer_Session_Active := TRUE;
END_IF;

// ------------------------------------------------------
// Peer lease validation foundation.
// ------------------------------------------------------

IF L_Peer_Session_Active THEN
    L_Delta_MS := L_Now_MS - GVL_DISTRIBUTED_EPOCH.Peer_Last_Refresh_MS;

    IF GVL_DISTRIBUTED_EPOCH.Peer_Lease_Active THEN
        IF L_Delta_MS > GVL_DISTRIBUTED_EPOCH.Peer_Lease_Timeout_MS THEN
            GVL_DISTRIBUTED_EPOCH.Peer_Lease_Expired := TRUE;

            L_Distributed_Valid := FALSE;
            L_Error_Code := 13000;
            L_Error_Text := 'Peer lease expired';
        END_IF;
    END_IF;
END_IF;

// ------------------------------------------------------
// Peer runtime continuity foundation.
// ------------------------------------------------------

IF L_Distributed_Valid AND L_Peer_Session_Active THEN
    IF GVL_DISTRIBUTED_EPOCH.Peer_Runtime_Epoch < GVL_DISTRIBUTED_EPOCH.Local_Runtime_Epoch THEN
        GVL_DISTRIBUTED_EPOCH.Peer_Runtime_Stale := TRUE;
    END_IF;
END_IF;

// ------------------------------------------------------
// Peer snapshot continuity foundation.
// ------------------------------------------------------

IF L_Distributed_Valid AND L_Peer_Session_Active THEN
    IF GVL_DISTRIBUTED_EPOCH.Peer_Snapshot_Epoch < GVL_DISTRIBUTED_EPOCH.Local_Snapshot_Epoch THEN
        GVL_DISTRIBUTED_EPOCH.Peer_Snapshot_Stale := TRUE;
    END_IF;
END_IF;

// ------------------------------------------------------
// Peer boot generation continuity foundation.
// ------------------------------------------------------

IF L_Distributed_Valid AND L_Peer_Session_Active THEN
    IF GVL_DISTRIBUTED_EPOCH.Peer_Boot_Generation <> GVL_DISTRIBUTED_EPOCH.Local_Boot_Generation THEN
        GVL_DISTRIBUTED_EPOCH.Peer_Boot_Mismatch := TRUE;
    END_IF;
END_IF;

// ------------------------------------------------------
// Peer fencing continuity foundation.
// ------------------------------------------------------

IF L_Distributed_Valid AND L_Peer_Session_Active THEN
    IF GVL_DISTRIBUTED_EPOCH.Peer_Fencing_Token = GVL_DISTRIBUTED_EPOCH.Local_Fencing_Token THEN
        GVL_DISTRIBUTED_EPOCH.Peer_Fencing_Conflict := TRUE;

        L_Distributed_Valid := FALSE;
        L_Error_Code := 13001;
        L_Error_Text := 'Peer fencing conflict detected';
    END_IF;
END_IF;

// ------------------------------------------------------
// Distributed semantic continuity.
// ------------------------------------------------------

IF GVL_DISTRIBUTED_EPOCH.Peer_Runtime_Stale
OR GVL_DISTRIBUTED_EPOCH.Peer_Snapshot_Stale
OR GVL_DISTRIBUTED_EPOCH.Peer_Boot_Mismatch
OR GVL_DISTRIBUTED_EPOCH.Peer_Fencing_Conflict
THEN
    GVL_DISTRIBUTED_EPOCH.Peer_Semantic_Continuity_Lost := TRUE;
END_IF;

// ------------------------------------------------------
// Publish distributed epoch state.
// ------------------------------------------------------

IF L_Distributed_Valid THEN
    GVL_DISTRIBUTED_EPOCH.Distributed_Epoch := GVL_DISTRIBUTED_EPOCH.Distributed_Epoch + 1;
    GVL_DISTRIBUTED_EPOCH.Distributed_Reconciliation_Epoch := GVL_DISTRIBUTED_EPOCH.Distributed_Reconciliation_Epoch + 1;

    GVL_DISTRIBUTED_EPOCH.Distributed_Epoch_Consistent := TRUE;
    GVL_DISTRIBUTED_EPOCH.Distributed_Reconciliation_Valid := TRUE;
    GVL_DISTRIBUTED_EPOCH.Distributed_Publication_Allowed := TRUE;

    GVL_DISTRIBUTED_EPOCH.Distributed_Quarantine_Active := FALSE;

    GVL_DISTRIBUTED_EPOCH.Peer_Last_Reconciliation_MS := L_Now_MS;

    GVL_DISTRIBUTED_EPOCH.Distributed_Last_Error_Code := 0;
    GVL_DISTRIBUTED_EPOCH.Distributed_Last_Error_Text := '';
ELSE
    GVL_DISTRIBUTED_EPOCH.Distributed_Epoch_Consistent := FALSE;
    GVL_DISTRIBUTED_EPOCH.Distributed_Reconciliation_Valid := FALSE;
    GVL_DISTRIBUTED_EPOCH.Distributed_Publication_Allowed := FALSE;

    GVL_DISTRIBUTED_EPOCH.Distributed_Quarantine_Active := TRUE;

    GVL_DISTRIBUTED_EPOCH.Distributed_Last_Error_Code := L_Error_Code;
    GVL_DISTRIBUTED_EPOCH.Distributed_Last_Error_Text := L_Error_Text;
END_IF;
END_PROGRAM

(* ---- PRG_Distributed_Peer_Ingestion.st ---- *)
PROGRAM PRG_Distributed_Peer_Ingestion
VAR
    L_Now_MS : UDINT;
END_VAR

// ======================================================
// DISTRIBUTED PEER INGESTION
// ======================================================
// Bounded peer-session ingestion layer.
//
// Purpose:
// normalize remote PLC liveness/session visibility into
// distributed peer-input fields consumed by distributed governors.
//
// This layer does NOT:
// - perform reconciliation/quarantine decisions
// - perform split-brain detection
// - validate peer publication correctness
// - mutate local runtime authority
//
// Current implementation status:
// peer epoch/token values are projected from currently available
// remote PLC runtime visibility until a richer transport/session
// contract is implemented.
// ======================================================

L_Now_MS := GVL_STATUS.G_System_Time_MS;

// ------------------------------------------------------
// Peer session freshness projection.
// ------------------------------------------------------

GVL_DISTRIBUTED_EPOCH.Peer_Last_Refresh_MS :=
    GVL_STATUS.G_Remote_PLC_Last_Seen_MS;

GVL_DISTRIBUTED_EPOCH.Peer_Lease_Active :=
    GVL_STATUS.G_Remote_PLC_Alive;

// ------------------------------------------------------
// Peer runtime visibility projection.
// ------------------------------------------------------

IF GVL_STATUS.G_Remote_PLC_Alive THEN
    // Transitional projection model:
    // until explicit remote epoch transport exists,
    // peer visibility mirrors current known remote-active session.

    GVL_DISTRIBUTED_EPOCH.Peer_Runtime_Epoch :=
        GVL_RUNTIME_EPOCH.Runtime_Epoch;

    GVL_DISTRIBUTED_EPOCH.Peer_Snapshot_Epoch :=
        GVL_RUNTIME_SNAPSHOT.Runtime_Snapshot_Epoch;

    GVL_DISTRIBUTED_EPOCH.Peer_Boot_Generation :=
        GVL_STATUS.G_Active_PLC_ID;

    // Transitional fencing projection.
    // Explicit remote fencing-token exchange is not yet implemented.
    GVL_DISTRIBUTED_EPOCH.Peer_Fencing_Token :=
        GVL_STATUS.G_Active_PLC_ID;
ELSE
    GVL_DISTRIBUTED_EPOCH.Peer_Lease_Active := FALSE;
END_IF;

// >>> BULK_SYNC_ANCHOR: PRG_Distributed_Peer_Ingestion <<<
END_PROGRAM

(* ---- PRG_Distributed_Runtime_Supervisor.st ---- *)
PROGRAM PRG_Distributed_Runtime_Supervisor
VAR
    fbClusterSafetyBarrier : FB_Cluster_Safety_Barrier_Runtime;

    fbRuntimeDiscovery : FB_Runtime_Node_Discovery;
    fbRuntimeSessions : FB_Runtime_Session_Governance;

    fbDistributedRuntimeContinuity : FB_Distributed_Runtime_Continuity;
    fbDistributedAuthority : FB_Distributed_Authority_Arbitration;

    fbRuntimeBusReplication : FB_Runtime_Bus_Replication;

    fbMQTTRuntimeAdapter : FB_MQTT_Runtime_Adapter;
    fbOPCUARuntimeAdapter : FB_OPCUA_Runtime_Adapter;
    fbADSRuntimeAdapter : FB_ADS_Runtime_Adapter;

    fbProjectionOwnership : FB_Distributed_Projection_Ownership_Runtime;
    fbDistributedOrchestration : FB_Distributed_Orchestration_Runtime;
    fbRecoveryLock : FB_Distributed_Recovery_Lock_Runtime;

    fbExecutionGates : FB_Distributed_Execution_Gates_Runtime;
    fbClusterRuntimeFSM : FB_Cluster_Runtime_FSM;
END_VAR

// Root distributed runtime execution chain.
//
// Execution order intentionally deterministic:
// safety -> discovery -> sessions -> authority -> replication
// -> transport -> ownership -> orchestration -> recovery locking
// -> unified execution gates -> cluster runtime FSM.
//
// Important convergence contract:
// execution gates must never reopen distributed execution authority
// before finalized convergence/publication continuity is achieved.
//
// Required finalized authority chain:
// immutable snapshot
// -> distributed reconciliation
// -> distributed commit continuity
// -> finalized publication validity
// -> convergence release
// -> execution gates reopen.

fbClusterSafetyBarrier(
    VI_Enable := TRUE,
    VI_System_Time_MS := GVL_STATUS.G_System_Time_MS
);

fbRuntimeDiscovery(
    VI_Enable := TRUE,
    VI_System_Time_MS := GVL_STATUS.G_System_Time_MS
);

fbRuntimeSessions(
    VI_Enable := TRUE,
    VI_System_Time_MS := GVL_STATUS.G_System_Time_MS
);

fbDistributedRuntimeContinuity(
    VI_Enable := TRUE,
    VI_System_Time_MS := GVL_STATUS.G_System_Time_MS
);

fbDistributedAuthority(
    VI_Enable := TRUE,
    VI_System_Time_MS := GVL_STATUS.G_System_Time_MS
);

fbRuntimeBusReplication(
    VI_Enable := TRUE,
    VI_System_Time_MS := GVL_STATUS.G_System_Time_MS
);

fbMQTTRuntimeAdapter(
    VI_Enable := TRUE,
    VI_System_Time_MS := GVL_STATUS.G_System_Time_MS
);

fbOPCUARuntimeAdapter(
    VI_Enable := TRUE,
    VI_System_Time_MS := GVL_STATUS.G_System_Time_MS
);

fbADSRuntimeAdapter(
    VI_Enable := TRUE,
    VI_System_Time_MS := GVL_STATUS.G_System_Time_MS
);

fbProjectionOwnership(
    VI_Enable := TRUE,
    VI_System_Time_MS := GVL_STATUS.G_System_Time_MS
);

fbDistributedOrchestration(
    VI_Enable := TRUE,
    VI_System_Time_MS := GVL_STATUS.G_System_Time_MS
);

fbRecoveryLock(
    VI_Enable := TRUE,
    VI_System_Time_MS := GVL_STATUS.G_System_Time_MS
);

fbExecutionGates(
    VI_Enable := TRUE,
    VI_System_Time_MS := GVL_STATUS.G_System_Time_MS
);

fbClusterRuntimeFSM(
    VI_Enable := TRUE,
    VI_System_Time_MS := GVL_STATUS.G_System_Time_MS
);

END_PROGRAM

(* ---- PRG_Distributed_Snapshot_Governor.st ---- *)
PROGRAM PRG_Distributed_Snapshot_Governor
VAR
    L_Now_MS : UDINT;
    L_Delta_MS : UDINT;
    L_Distributed_Snapshot_Valid : BOOL := TRUE;
    L_Error_Code : UDINT := 0;
    L_Error_Text : STRING(160) := '';
    L_Peer_Session_Active : BOOL := FALSE;
END_VAR

L_Now_MS := GVL_STATUS.G_System_Time_MS;
L_Distributed_Snapshot_Valid := TRUE;
L_Error_Code := 0;
L_Error_Text := '';

// ======================================================
// DISTRIBUTED IMMUTABLE SNAPSHOT GOVERNOR
// ======================================================
// Governs immutable peer publication snapshot exchange.
// Publication-authoritative only.
// Does not invalidate runtime barrier, PLC fencing
// or local immutable snapshot freeze.
//
// Current implementation mode:
// peer-optional foundation mode.
//
// Missing peer topology is NOT treated as divergence.
// Peer validation activates only after real peer
// synchronization state exists.
// ======================================================

GVL_DISTRIBUTED_SNAPSHOT.Peer_Publication_Stale := FALSE;
GVL_DISTRIBUTED_SNAPSHOT.Peer_Snapshot_Not_Immutable := FALSE;
GVL_DISTRIBUTED_SNAPSHOT.Peer_Publication_Divergence := FALSE;
GVL_DISTRIBUTED_SNAPSHOT.Peer_Publication_Reconciliation_Lost := FALSE;
GVL_DISTRIBUTED_SNAPSHOT.Peer_Snapshot_Lease_Expired := FALSE;

// ------------------------------------------------------
// Local immutable publication projection.
// ------------------------------------------------------

GVL_DISTRIBUTED_SNAPSHOT.Local_Distributed_Snapshot_Epoch := GVL_DISTRIBUTED_SNAPSHOT.Distributed_Snapshot_Epoch;
GVL_DISTRIBUTED_SNAPSHOT.Local_Runtime_Snapshot_Epoch := GVL_RUNTIME_SNAPSHOT.Snapshot_Epoch;
GVL_DISTRIBUTED_SNAPSHOT.Local_Publication_Epoch := GVL_OUTPUT_EPOCH.Output_Publication_Epoch;

// ------------------------------------------------------
// Local immutable publication freeze semantics.
// ------------------------------------------------------

IF GVL_RUNTIME_SNAPSHOT.Snapshot_Frozen
AND GVL_RUNTIME_SNAPSHOT.Snapshot_Publication_Allowed
AND GVL_RUNTIME_SNAPSHOT.Snapshot_Copy_Valid
AND GVL_RUNTIME_SNAPSHOT.Snapshot_Isolation_Valid
THEN
    GVL_DISTRIBUTED_SNAPSHOT.Distributed_Snapshot_Frozen := TRUE;
ELSE
    GVL_DISTRIBUTED_SNAPSHOT.Distributed_Snapshot_Frozen := FALSE;

    L_Distributed_Snapshot_Valid := FALSE;
    L_Error_Code := 14000;
    L_Error_Text := 'Local immutable snapshot not frozen';
END_IF;

// ------------------------------------------------------
// Peer session detection.
// ------------------------------------------------------

IF GVL_DISTRIBUTED_SNAPSHOT.Peer_Publication_Epoch > 0 THEN
    L_Peer_Session_Active := TRUE;
END_IF;

IF GVL_DISTRIBUTED_SNAPSHOT.Peer_Runtime_Snapshot_Epoch > 0 THEN
    L_Peer_Session_Active := TRUE;
END_IF;

IF GVL_DISTRIBUTED_SNAPSHOT.Peer_Distributed_Snapshot_Epoch > 0 THEN
    L_Peer_Session_Active := TRUE;
END_IF;

IF GVL_DISTRIBUTED_SNAPSHOT.Peer_Snapshot_Immutable THEN
    L_Peer_Session_Active := TRUE;
END_IF;

// ------------------------------------------------------
// Peer snapshot lease validation.
// ------------------------------------------------------

IF L_Distributed_Snapshot_Valid AND L_Peer_Session_Active THEN
    L_Delta_MS := L_Now_MS - GVL_DISTRIBUTED_SNAPSHOT.Peer_Snapshot_Last_Refresh_MS;

    IF GVL_DISTRIBUTED_SNAPSHOT.Peer_Snapshot_Lease_Active THEN
        IF L_Delta_MS > GVL_DISTRIBUTED_SNAPSHOT.Peer_Snapshot_Lease_Timeout_MS THEN
            GVL_DISTRIBUTED_SNAPSHOT.Peer_Snapshot_Lease_Expired := TRUE;

            L_Distributed_Snapshot_Valid := FALSE;
            L_Error_Code := 14001;
            L_Error_Text := 'Peer snapshot lease expired';
        END_IF;
    END_IF;
END_IF;

// ------------------------------------------------------
// Peer immutable snapshot semantics.
// ------------------------------------------------------

IF L_Distributed_Snapshot_Valid AND L_Peer_Session_Active THEN
    IF NOT GVL_DISTRIBUTED_SNAPSHOT.Peer_Snapshot_Immutable THEN
        GVL_DISTRIBUTED_SNAPSHOT.Peer_Snapshot_Not_Immutable := TRUE;

        L_Distributed_Snapshot_Valid := FALSE;
        L_Error_Code := 14002;
        L_Error_Text := 'Peer snapshot not immutable';
    END_IF;
END_IF;

// ------------------------------------------------------
// Peer publication continuity.
// ------------------------------------------------------

IF L_Distributed_Snapshot_Valid AND L_Peer_Session_Active THEN
    IF GVL_DISTRIBUTED_SNAPSHOT.Peer_Publication_Epoch < GVL_DISTRIBUTED_SNAPSHOT.Local_Publication_Epoch THEN
        GVL_DISTRIBUTED_SNAPSHOT.Peer_Publication_Stale := TRUE;
    END_IF;
END_IF;

// ------------------------------------------------------
// Peer publication reconciliation continuity.
// ------------------------------------------------------

IF L_Distributed_Snapshot_Valid AND L_Peer_Session_Active THEN
    IF GVL_DISTRIBUTED_SNAPSHOT.Peer_Runtime_Snapshot_Epoch <> GVL_DISTRIBUTED_SNAPSHOT.Local_Runtime_Snapshot_Epoch THEN
        GVL_DISTRIBUTED_SNAPSHOT.Peer_Publication_Divergence := TRUE;
    END_IF;
END_IF;

IF GVL_DISTRIBUTED_SNAPSHOT.Peer_Publication_Stale
OR GVL_DISTRIBUTED_SNAPSHOT.Peer_Publication_Divergence
OR GVL_DISTRIBUTED_SNAPSHOT.Peer_Snapshot_Not_Immutable
THEN
    GVL_DISTRIBUTED_SNAPSHOT.Peer_Publication_Reconciliation_Lost := TRUE;
END_IF;

// ------------------------------------------------------
// Publish authoritative distributed snapshot state.
// ------------------------------------------------------

IF L_Distributed_Snapshot_Valid THEN
    GVL_DISTRIBUTED_SNAPSHOT.Distributed_Snapshot_Epoch := GVL_DISTRIBUTED_SNAPSHOT.Distributed_Snapshot_Epoch + 1;
    GVL_DISTRIBUTED_SNAPSHOT.Distributed_Snapshot_Reconciliation_Epoch := GVL_DISTRIBUTED_SNAPSHOT.Distributed_Snapshot_Reconciliation_Epoch + 1;

    GVL_DISTRIBUTED_SNAPSHOT.Distributed_Publication_Reconciled := TRUE;
    GVL_DISTRIBUTED_SNAPSHOT.Distributed_Publication_Freeze_Valid := TRUE;
    GVL_DISTRIBUTED_SNAPSHOT.Distributed_Snapshot_Consistent := TRUE;

    GVL_DISTRIBUTED_SNAPSHOT.Distributed_Snapshot_Quarantine_Active := FALSE;

    GVL_DISTRIBUTED_SNAPSHOT.Distributed_Snapshot_Last_Error_Code := 0;
    GVL_DISTRIBUTED_SNAPSHOT.Distributed_Snapshot_Last_Error_Text := '';
ELSE
    GVL_DISTRIBUTED_SNAPSHOT.Distributed_Publication_Reconciled := FALSE;
    GVL_DISTRIBUTED_SNAPSHOT.Distributed_Publication_Freeze_Valid := FALSE;
    GVL_DISTRIBUTED_SNAPSHOT.Distributed_Snapshot_Consistent := FALSE;

    GVL_DISTRIBUTED_SNAPSHOT.Distributed_Snapshot_Quarantine_Active := TRUE;

    GVL_DISTRIBUTED_SNAPSHOT.Distributed_Snapshot_Last_Error_Code := L_Error_Code;
    GVL_DISTRIBUTED_SNAPSHOT.Distributed_Snapshot_Last_Error_Text := L_Error_Text;
END_IF;
END_PROGRAM

(* ---- PRG_Distributed_Snapshot_Publication.st ---- *)
PROGRAM PRG_Distributed_Snapshot_Publication
// ======================================================
// DISTRIBUTED SNAPSHOT PUBLICATION
// ======================================================
// Canonical local distributed snapshot export into the
// HA replication boundary.
//
// Purpose:
// publish normalized immutable snapshot/publication state
// into the dedicated HA boundary before snapshot ingestion.
//
// This layer does NOT:
// - perform reconciliation
// - validate peer snapshot state
// - arbitrate distributed publication authority
//
// Disabled HA replication must not leave stale snapshot mirrors.
// ======================================================

IF NOT GVL_HA_SESSION_REPLICATION.HA_Replication_Enabled THEN
    GVL_HA_SESSION_REPLICATION.HA_Remote_Distributed_Snapshot_Epoch := 0;
    GVL_HA_SESSION_REPLICATION.HA_Remote_Runtime_Snapshot_Epoch := 0;
    GVL_HA_SESSION_REPLICATION.HA_Remote_Publication_Epoch := 0;
    GVL_HA_SESSION_REPLICATION.HA_Remote_Snapshot_Immutable := FALSE;
    GVL_HA_SESSION_REPLICATION.HA_Remote_Snapshot_Last_Refresh_MS := 0;
    RETURN;
END_IF;

GVL_HA_SESSION_REPLICATION.HA_Remote_Distributed_Snapshot_Epoch :=
    GVL_DISTRIBUTED_SNAPSHOT.Local_Distributed_Snapshot_Epoch;

GVL_HA_SESSION_REPLICATION.HA_Remote_Runtime_Snapshot_Epoch :=
    GVL_RUNTIME_SNAPSHOT.Snapshot_Epoch;

GVL_HA_SESSION_REPLICATION.HA_Remote_Publication_Epoch :=
    GVL_RUNTIME_SNAPSHOT.Snapshot_Publication_Epoch;

GVL_HA_SESSION_REPLICATION.HA_Remote_Snapshot_Immutable :=
    GVL_RUNTIME_SNAPSHOT.Snapshot_Frozen
    AND GVL_RUNTIME_SNAPSHOT.Snapshot_Publication_Allowed
    AND GVL_RUNTIME_SNAPSHOT.Snapshot_Copy_Valid
    AND GVL_RUNTIME_SNAPSHOT.Snapshot_Isolation_Valid;

GVL_HA_SESSION_REPLICATION.HA_Remote_Snapshot_Last_Refresh_MS :=
    GVL_STATUS.G_System_Time_MS;

// >>> BULK_SYNC_ANCHOR: PRG_Distributed_Snapshot_Publication <<<
END_PROGRAM

(* ---- PRG_Domain_Execution_Policy.st ---- *)
PROGRAM PRG_Domain_Execution_Policy
// Observational domain execution policy.
// Classifies domains as critical, periodic or idle-by-design.
// Does not gate execution and does not write physical outputs.
VAR
    L_i : INT;
    L_Heating_Output_Active : BOOL;
    L_Vent_Output_Active : BOOL;
END_VAR

GVL_DOMAIN_EXECUTION_POLICY.G_Last_Update_MS := GVL_TIME_SERVICE.G_Now_MS;

GVL_DOMAIN_EXECUTION_POLICY.G_Security_Context_Active :=
    GVL_ALARM.G_Security_Armed
    OR GVL_ALARM.G_Security_Alarm;

GVL_DOMAIN_EXECUTION_POLICY.G_Away_Context_Active :=
    GVL_STATUS.G_Current_Scenario = SCENARIO_AWAY;

GVL_DOMAIN_EXECUTION_POLICY.G_Presence_Context_Active :=
    GVL_STATUS.G_Current_Scenario = SCENARIO_PRESENCE;

GVL_DOMAIN_EXECUTION_POLICY.G_Emergency_Context_Active :=
    (GVL_SAFETY_SHUTDOWN.G_Safety_Mode = FIRE)
    OR (GVL_SAFETY_SHUTDOWN.G_Safety_Mode = GAS)
    OR (GVL_SAFETY_SHUTDOWN.G_Safety_Mode = WATER_LEAK)
    OR (GVL_SAFETY_SHUTDOWN.G_Safety_Mode = GLOBAL_STOP);

// ------------------------------------------------------------------------------
// Access policy.
// Critical when emergency semantics or an access command/pulse is active.
// Periodic when security/away context is active, even without a current pulse.
// ------------------------------------------------------------------------------
GVL_DOMAIN_EXECUTION_POLICY.Access_Critical_Run :=
    (GVL_SAFETY_SHUTDOWN.G_Safety_Mode = FIRE)
    OR (GVL_SAFETY_SHUTDOWN.G_Safety_Mode = GAS)
    OR GVL_COMMAND_SHADOW.G_Lock_1_Open
    OR GVL_COMMAND_SHADOW.G_Lock_1_Close
    OR GVL_COMMAND_SHADOW.G_Lock_2_Open
    OR GVL_COMMAND_SHADOW.G_Lock_2_Close
    OR GVL_COMMAND_SHADOW.G_Gate_Open
    OR GVL_COMMAND_SHADOW.G_Wicket_Open
    OR GVL_ACCESS_RUNTIME.G_Any_Pulse_Active;

GVL_DOMAIN_EXECUTION_POLICY.Access_Periodic_Run :=
    (NOT GVL_DOMAIN_EXECUTION_POLICY.Access_Critical_Run)
    AND (
        GVL_DOMAIN_EXECUTION_POLICY.G_Security_Context_Active
        OR GVL_DOMAIN_EXECUTION_POLICY.G_Away_Context_Active
    );

GVL_DOMAIN_EXECUTION_POLICY.Access_Idle_By_Design :=
    NOT GVL_DOMAIN_EXECUTION_POLICY.Access_Critical_Run
    AND NOT GVL_DOMAIN_EXECUTION_POLICY.Access_Periodic_Run;

IF GVL_DOMAIN_EXECUTION_POLICY.Access_Critical_Run THEN
    GVL_DOMAIN_EXECUTION_POLICY.Access_Mode := 2;
ELSIF GVL_DOMAIN_EXECUTION_POLICY.Access_Periodic_Run THEN
    GVL_DOMAIN_EXECUTION_POLICY.Access_Mode := 1;
ELSE
    GVL_DOMAIN_EXECUTION_POLICY.Access_Mode := 0;
END_IF;

// ------------------------------------------------------------------------------
// Lighting policy.
// Critical for fire/evacuation/security alarm/active outputs.
// Periodic for security armed / away / presence scenarios.
// ------------------------------------------------------------------------------
GVL_DOMAIN_EXECUTION_POLICY.Lighting_Critical_Run :=
    (GVL_SAFETY_SHUTDOWN.G_Safety_Mode = FIRE)
    OR GVL_STATE.G_Evacuation_Lighting_Active
    OR GVL_LIGHTING_RUNTIME.G_Emergency_Override_Active
    OR GVL_LIGHTING_RUNTIME.G_Any_Light_Active
    OR GVL_LIGHTING_RUNTIME.G_Any_Blind_Not_Safe_Open
    OR GVL_LIGHTING_RUNTIME.G_Any_Socket_Active
    OR GVL_ALARM.G_Security_Alarm;

GVL_DOMAIN_EXECUTION_POLICY.Lighting_Periodic_Run :=
    (NOT GVL_DOMAIN_EXECUTION_POLICY.Lighting_Critical_Run)
    AND (
        GVL_DOMAIN_EXECUTION_POLICY.G_Security_Context_Active
        OR GVL_DOMAIN_EXECUTION_POLICY.G_Away_Context_Active
        OR GVL_DOMAIN_EXECUTION_POLICY.G_Presence_Context_Active
    );

GVL_DOMAIN_EXECUTION_POLICY.Lighting_Idle_By_Design :=
    NOT GVL_DOMAIN_EXECUTION_POLICY.Lighting_Critical_Run
    AND NOT GVL_DOMAIN_EXECUTION_POLICY.Lighting_Periodic_Run;

IF GVL_DOMAIN_EXECUTION_POLICY.Lighting_Critical_Run THEN
    GVL_DOMAIN_EXECUTION_POLICY.Lighting_Mode := 2;
ELSIF GVL_DOMAIN_EXECUTION_POLICY.Lighting_Periodic_Run THEN
    GVL_DOMAIN_EXECUTION_POLICY.Lighting_Mode := 1;
ELSE
    GVL_DOMAIN_EXECUTION_POLICY.Lighting_Mode := 0;
END_IF;

// ------------------------------------------------------------------------------
// Water policy.
// Critical when leak/global path/output close/recovery is active.
// Periodic when water status has no demand but system is in security/away context.
// ------------------------------------------------------------------------------
GVL_DOMAIN_EXECUTION_POLICY.Water_Critical_Run :=
    (GVL_SAFETY_SHUTDOWN.G_Safety_Mode = WATER_LEAK)
    OR GVL_COMMAND_SHADOW.G_Water_Block
    OR GVL_COMMAND_SHADOW.G_Water_Emergency_Stop
    OR GVL_COMMAND_SHADOW.G_Close_Valve_35
    OR GVL_COMMAND_SHADOW.G_Close_Valve_36
    OR GVL_WATER_DOMAIN_STATUS.G_Recovery_Requested
    OR GVL_WATER_DOMAIN_STATUS.G_Global_Path_Active
    OR GVL_WATER_DOMAIN_STATUS.G_Output_35_Active
    OR GVL_WATER_DOMAIN_STATUS.G_Output_36_Active
    OR GVL_WATER_DOMAIN_STATUS.G_Any_Zone_Active;

GVL_DOMAIN_EXECUTION_POLICY.Water_Periodic_Run :=
    (NOT GVL_DOMAIN_EXECUTION_POLICY.Water_Critical_Run)
    AND (
        GVL_DOMAIN_EXECUTION_POLICY.G_Security_Context_Active
        OR GVL_DOMAIN_EXECUTION_POLICY.G_Away_Context_Active
    );

GVL_DOMAIN_EXECUTION_POLICY.Water_Idle_By_Design :=
    NOT GVL_DOMAIN_EXECUTION_POLICY.Water_Critical_Run
    AND NOT GVL_DOMAIN_EXECUTION_POLICY.Water_Periodic_Run;

IF GVL_DOMAIN_EXECUTION_POLICY.Water_Critical_Run THEN
    GVL_DOMAIN_EXECUTION_POLICY.Water_Mode := 2;
ELSIF GVL_DOMAIN_EXECUTION_POLICY.Water_Periodic_Run THEN
    GVL_DOMAIN_EXECUTION_POLICY.Water_Mode := 1;
ELSE
    GVL_DOMAIN_EXECUTION_POLICY.Water_Mode := 0;
END_IF;

// ------------------------------------------------------------------------------
// Heating policy.
// Critical for emergency/freeze/gas/DHW/active outputs.
// Periodic for comfort scenarios or low-demand normal supervision.
// ------------------------------------------------------------------------------
L_Heating_Output_Active :=
    GVL_HEATING_OUTPUT.DO_DHW_Heating_Pump
    OR GVL_HEATING_OUTPUT.DO_DHW_Circ_Pump
    OR GVL_HEATING_OUTPUT.DO_Backup_Circulation_Pump
    OR GVL_HEATING_OUTPUT.DO_Electric_Heater_Enable;

FOR L_i := 1 TO GVL_CONSTANTS.C_MAX_HEATING_CIRCUITS DO
    L_Heating_Output_Active :=
        L_Heating_Output_Active
        OR GVL_HEATING_OUTPUT.DO_Zone_Valves[L_i];
END_FOR;

FOR L_i := 1 TO GVL_CONSTANTS.C_MAX_MANIFOLDS DO
    L_Heating_Output_Active :=
        L_Heating_Output_Active
        OR GVL_HEATING_OUTPUT.DO_Manifold_Pumps[L_i]
        OR (GVL_HEATING_OUTPUT.AO_Manifold_Valves[L_i] > 0);
END_FOR;

GVL_DOMAIN_EXECUTION_POLICY.Heating_Critical_Run :=
    GVL_COMMAND_SHADOW.G_Heating_Emergency_Stop
    OR GVL_COMMAND_SHADOW.G_Heating_Gas_Safety_Stop
    OR GVL_STATE.G_Safety_Gas_Latched
    OR GVL_STATE.G_Safety_Freeze_Risk
    OR L_Heating_Output_Active;

GVL_DOMAIN_EXECUTION_POLICY.Heating_Periodic_Run :=
    (NOT GVL_DOMAIN_EXECUTION_POLICY.Heating_Critical_Run)
    AND (
        GVL_STATUS.G_Current_Scenario = SCENARIO_MORNING
        OR GVL_STATUS.G_Current_Scenario = SCENARIO_EVENING
        OR GVL_STATUS.G_Current_Scenario = SCENARIO_SLEEP
        OR GVL_STATUS.G_Current_Scenario = SCENARIO_PRESENCE
        OR GVL_INPUT.IN_Preheat_Request
        OR GVL_INPUT.IN_Freeze_Request
    );

GVL_DOMAIN_EXECUTION_POLICY.Heating_Idle_By_Design :=
    NOT GVL_DOMAIN_EXECUTION_POLICY.Heating_Critical_Run
    AND NOT GVL_DOMAIN_EXECUTION_POLICY.Heating_Periodic_Run;

IF GVL_DOMAIN_EXECUTION_POLICY.Heating_Critical_Run THEN
    GVL_DOMAIN_EXECUTION_POLICY.Heating_Mode := 2;
ELSIF GVL_DOMAIN_EXECUTION_POLICY.Heating_Periodic_Run THEN
    GVL_DOMAIN_EXECUTION_POLICY.Heating_Mode := 1;
ELSE
    GVL_DOMAIN_EXECUTION_POLICY.Heating_Mode := 0;
END_IF;

// ------------------------------------------------------------------------------
// Ventilation policy.
// Critical for gas/fire/smoke/emergency boost or active outputs.
// Periodic for occupancy/away/presence/background air-quality supervision.
// ------------------------------------------------------------------------------
L_Vent_Output_Active := GVL_VENT_OUTPUT.DO_Vent_Enable;

FOR L_i := 1 TO GVL_CONSTANTS.C_MAX_SUPPLY_FANS DO
    L_Vent_Output_Active :=
        L_Vent_Output_Active
        OR (GVL_VENT_OUTPUT.AO_Supply_Fans[L_i] > 0);
END_FOR;

FOR L_i := 1 TO GVL_CONSTANTS.C_MAX_EXHAUST_FANS DO
    L_Vent_Output_Active :=
        L_Vent_Output_Active
        OR (GVL_VENT_OUTPUT.AO_Exhaust_Fans[L_i] > 0);
END_FOR;

GVL_DOMAIN_EXECUTION_POLICY.Vent_Critical_Run :=
    (GVL_SAFETY_SHUTDOWN.G_Safety_Mode = FIRE)
    OR (GVL_SAFETY_SHUTDOWN.G_Safety_Mode = GAS)
    OR GVL_COMMAND_SHADOW.G_Vent_PV3_Boost
    OR GVL_COMMAND_SHADOW.G_Exhaust_100_Req
    OR GVL_COMMAND_SHADOW.G_Vent_Smoke_Exhaust
    OR L_Vent_Output_Active;

GVL_DOMAIN_EXECUTION_POLICY.Vent_Periodic_Run :=
    (NOT GVL_DOMAIN_EXECUTION_POLICY.Vent_Critical_Run)
    AND (
        GVL_DOMAIN_EXECUTION_POLICY.G_Presence_Context_Active
        OR GVL_DOMAIN_EXECUTION_POLICY.G_Away_Context_Active
        OR GVL_INTENT_BEHAVIOR.I_Request_Ventilation_Boost
    );

GVL_DOMAIN_EXECUTION_POLICY.Vent_Idle_By_Design :=
    NOT GVL_DOMAIN_EXECUTION_POLICY.Vent_Critical_Run
    AND NOT GVL_DOMAIN_EXECUTION_POLICY.Vent_Periodic_Run;

IF GVL_DOMAIN_EXECUTION_POLICY.Vent_Critical_Run THEN
    GVL_DOMAIN_EXECUTION_POLICY.Vent_Mode := 2;
ELSIF GVL_DOMAIN_EXECUTION_POLICY.Vent_Periodic_Run THEN
    GVL_DOMAIN_EXECUTION_POLICY.Vent_Mode := 1;
ELSE
    GVL_DOMAIN_EXECUTION_POLICY.Vent_Mode := 0;
END_IF;

// ------------------------------------------------------------------------------
// Simulation policy.
// Runs only when enabled and there is test/security/away/presence context.
// ------------------------------------------------------------------------------
GVL_DOMAIN_EXECUTION_POLICY.Simulation_Context_Active :=
    GVL_SIMULATION.G_Test_Scenario_Active
    OR GVL_SIMULATION.G_Test_Start
    OR GVL_DOMAIN_EXECUTION_POLICY.G_Security_Context_Active
    OR GVL_DOMAIN_EXECUTION_POLICY.G_Away_Context_Active
    OR GVL_DOMAIN_EXECUTION_POLICY.G_Presence_Context_Active;

GVL_DOMAIN_EXECUTION_POLICY.Simulation_Run_Allowed :=
    GVL_SIMULATION.G_Simulation_Enable
    AND GVL_DOMAIN_EXECUTION_POLICY.Simulation_Context_Active
    AND NOT GVL_FABRIC_LIFECYCLE_REGISTRY.Simulation_Suspension_Recommended;

GVL_DOMAIN_EXECUTION_POLICY.Simulation_Idle_By_Design :=
    NOT GVL_DOMAIN_EXECUTION_POLICY.Simulation_Run_Allowed;

IF GVL_DOMAIN_EXECUTION_POLICY.Simulation_Run_Allowed THEN
    GVL_DOMAIN_EXECUTION_POLICY.Simulation_Mode := 1;
ELSE
    GVL_DOMAIN_EXECUTION_POLICY.Simulation_Mode := 0;
END_IF;

// ------------------------------------------------------------------------------
// Summary.
// ------------------------------------------------------------------------------
GVL_DOMAIN_EXECUTION_POLICY.Any_Critical_Run :=
    GVL_DOMAIN_EXECUTION_POLICY.Access_Critical_Run
    OR GVL_DOMAIN_EXECUTION_POLICY.Lighting_Critical_Run
    OR GVL_DOMAIN_EXECUTION_POLICY.Water_Critical_Run
    OR GVL_DOMAIN_EXECUTION_POLICY.Heating_Critical_Run
    OR GVL_DOMAIN_EXECUTION_POLICY.Vent_Critical_Run;

GVL_DOMAIN_EXECUTION_POLICY.Any_Periodic_Run :=
    GVL_DOMAIN_EXECUTION_POLICY.Access_Periodic_Run
    OR GVL_DOMAIN_EXECUTION_POLICY.Lighting_Periodic_Run
    OR GVL_DOMAIN_EXECUTION_POLICY.Water_Periodic_Run
    OR GVL_DOMAIN_EXECUTION_POLICY.Heating_Periodic_Run
    OR GVL_DOMAIN_EXECUTION_POLICY.Vent_Periodic_Run;

GVL_DOMAIN_EXECUTION_POLICY.Any_Idle_By_Design :=
    GVL_DOMAIN_EXECUTION_POLICY.Access_Idle_By_Design
    OR GVL_DOMAIN_EXECUTION_POLICY.Lighting_Idle_By_Design
    OR GVL_DOMAIN_EXECUTION_POLICY.Water_Idle_By_Design
    OR GVL_DOMAIN_EXECUTION_POLICY.Heating_Idle_By_Design
    OR GVL_DOMAIN_EXECUTION_POLICY.Vent_Idle_By_Design
    OR GVL_DOMAIN_EXECUTION_POLICY.Simulation_Idle_By_Design;

IF GVL_DOMAIN_EXECUTION_POLICY.Any_Critical_Run THEN
    GVL_DOMAIN_EXECUTION_POLICY.Status_Code := 2;
    GVL_DOMAIN_EXECUTION_POLICY.Status_Text := 'Domain execution policy critical activity present';
ELSIF GVL_DOMAIN_EXECUTION_POLICY.Any_Periodic_Run THEN
    GVL_DOMAIN_EXECUTION_POLICY.Status_Code := 1;
    GVL_DOMAIN_EXECUTION_POLICY.Status_Text := 'Domain execution policy periodic activity present';
ELSE
    GVL_DOMAIN_EXECUTION_POLICY.Status_Code := 0;
    GVL_DOMAIN_EXECUTION_POLICY.Status_Text := 'Domain execution policy idle by design';
END_IF;

// >>> BULK_SYNC_ANCHOR: PRG_Domain_Execution_Policy <<<
END_PROGRAM

(* ---- PRG_Domain_Execution_Policy_Periodic.st ---- *)
PROGRAM PRG_Domain_Execution_Policy_Periodic
// Observational periodic due gates for domain execution policy.
// Does not gate execution and does not write physical outputs.
VAR
    fbAccessDue : FB_Periodic_Due_Gate;
    fbLightingDue : FB_Periodic_Due_Gate;
    fbWaterDue : FB_Periodic_Due_Gate;
    fbHeatingDue : FB_Periodic_Due_Gate;
    fbVentDue : FB_Periodic_Due_Gate;
    fbSimulationDue : FB_Periodic_Due_Gate;
END_VAR

fbAccessDue(
    VI_Enable := GVL_DOMAIN_EXECUTION_POLICY.Access_Periodic_Run,
    VI_Now_MS := GVL_TIME_SERVICE.G_Now_MS,
    VI_Interval_MS := GVL_DOMAIN_EXECUTION_POLICY.Access_Periodic_Interval_MS
);
GVL_DOMAIN_EXECUTION_POLICY.Access_Periodic_Due := fbAccessDue.VO_Due;

fbLightingDue(
    VI_Enable := GVL_DOMAIN_EXECUTION_POLICY.Lighting_Periodic_Run,
    VI_Now_MS := GVL_TIME_SERVICE.G_Now_MS,
    VI_Interval_MS := GVL_DOMAIN_EXECUTION_POLICY.Lighting_Periodic_Interval_MS
);
GVL_DOMAIN_EXECUTION_POLICY.Lighting_Periodic_Due := fbLightingDue.VO_Due;

fbWaterDue(
    VI_Enable := GVL_DOMAIN_EXECUTION_POLICY.Water_Periodic_Run,
    VI_Now_MS := GVL_TIME_SERVICE.G_Now_MS,
    VI_Interval_MS := GVL_DOMAIN_EXECUTION_POLICY.Water_Periodic_Interval_MS
);
GVL_DOMAIN_EXECUTION_POLICY.Water_Periodic_Due := fbWaterDue.VO_Due;

fbHeatingDue(
    VI_Enable := GVL_DOMAIN_EXECUTION_POLICY.Heating_Periodic_Run,
    VI_Now_MS := GVL_TIME_SERVICE.G_Now_MS,
    VI_Interval_MS := GVL_DOMAIN_EXECUTION_POLICY.Heating_Periodic_Interval_MS
);
GVL_DOMAIN_EXECUTION_POLICY.Heating_Periodic_Due := fbHeatingDue.VO_Due;

fbVentDue(
    VI_Enable := GVL_DOMAIN_EXECUTION_POLICY.Vent_Periodic_Run,
    VI_Now_MS := GVL_TIME_SERVICE.G_Now_MS,
    VI_Interval_MS := GVL_DOMAIN_EXECUTION_POLICY.Vent_Periodic_Interval_MS
);
GVL_DOMAIN_EXECUTION_POLICY.Vent_Periodic_Due := fbVentDue.VO_Due;

fbSimulationDue(
    VI_Enable := GVL_DOMAIN_EXECUTION_POLICY.Simulation_Run_Allowed,
    VI_Now_MS := GVL_TIME_SERVICE.G_Now_MS,
    VI_Interval_MS := GVL_DOMAIN_EXECUTION_POLICY.Simulation_Periodic_Interval_MS
);
GVL_DOMAIN_EXECUTION_POLICY.Simulation_Periodic_Due := fbSimulationDue.VO_Due;

GVL_DOMAIN_EXECUTION_POLICY.Any_Periodic_Due :=
    GVL_DOMAIN_EXECUTION_POLICY.Access_Periodic_Due
    OR GVL_DOMAIN_EXECUTION_POLICY.Lighting_Periodic_Due
    OR GVL_DOMAIN_EXECUTION_POLICY.Water_Periodic_Due
    OR GVL_DOMAIN_EXECUTION_POLICY.Heating_Periodic_Due
    OR GVL_DOMAIN_EXECUTION_POLICY.Vent_Periodic_Due
    OR GVL_DOMAIN_EXECUTION_POLICY.Simulation_Periodic_Due;

// >>> BULK_SYNC_ANCHOR: PRG_Domain_Execution_Policy_Periodic <<<
END_PROGRAM

(* ---- PRG_Domain_Execution_Validation.st ---- *)
PROGRAM PRG_Domain_Execution_Validation
// Observational validation for policy-gated domain execution.
// Detects stale-output risks when a domain is classified idle.
VAR
    L_i : INT;
    L_Access_Output_Active : BOOL;
    L_Lighting_Output_Active : BOOL;
    L_Water_Output_Active : BOOL;
    L_Heating_Output_Active : BOOL;
    L_Vent_Output_Active : BOOL;
END_VAR

GVL_DOMAIN_EXECUTION_VALIDATION.G_Last_Update_MS := GVL_TIME_SERVICE.G_Now_MS;
GVL_DOMAIN_EXECUTION_VALIDATION.G_Validation_Executed := TRUE;
GVL_DOMAIN_EXECUTION_VALIDATION.G_Validation_Valid := TRUE;

L_Access_Output_Active :=
    GVL_ACCESS_OUTPUT.DO_Lock_1_Open
    OR GVL_ACCESS_OUTPUT.DO_Lock_1_Close
    OR GVL_ACCESS_OUTPUT.DO_Lock_2_Open
    OR GVL_ACCESS_OUTPUT.DO_Lock_2_Close
    OR GVL_ACCESS_OUTPUT.DO_Gate_Open
    OR GVL_ACCESS_OUTPUT.DO_Wicket_Open;

L_Lighting_Output_Active := FALSE;
FOR L_i := 1 TO GVL_CONSTANTS.C_MAX_LIGHT_ZONES DO
    L_Lighting_Output_Active :=
        L_Lighting_Output_Active
        OR (GVL_LIGHTING_OUTPUT.AO_Lighting_Levels[L_i] > 0);
END_FOR;
FOR L_i := 1 TO GVL_CONSTANTS.C_MAX_BLINDS DO
    L_Lighting_Output_Active :=
        L_Lighting_Output_Active
        OR (GVL_LIGHTING_OUTPUT.AO_Blinds_Positions[L_i] < 1000);
END_FOR;
FOR L_i := 1 TO GVL_CONSTANTS.C_MAX_SOCKETS DO
    L_Lighting_Output_Active :=
        L_Lighting_Output_Active
        OR GVL_LIGHTING_OUTPUT.DO_Sockets[L_i];
END_FOR;

L_Water_Output_Active :=
    GVL_WATER_OUTPUT.DO_Water_Valve_35_Close
    OR GVL_WATER_OUTPUT.DO_Water_Valve_36_Close;
FOR L_i := 1 TO GVL_CONSTANTS.C_MAX_WATER_ZONES DO
    L_Water_Output_Active :=
        L_Water_Output_Active
        OR GVL_WATER_OUTPUT.DO_Water_Zone_Enable[L_i];
END_FOR;

L_Heating_Output_Active :=
    GVL_HEATING_OUTPUT.DO_DHW_Heating_Pump
    OR GVL_HEATING_OUTPUT.DO_DHW_Circ_Pump
    OR GVL_HEATING_OUTPUT.DO_Backup_Circulation_Pump
    OR GVL_HEATING_OUTPUT.DO_Electric_Heater_Enable;
FOR L_i := 1 TO GVL_CONSTANTS.C_MAX_HEATING_CIRCUITS DO
    L_Heating_Output_Active :=
        L_Heating_Output_Active
        OR GVL_HEATING_OUTPUT.DO_Zone_Valves[L_i];
END_FOR;
FOR L_i := 1 TO GVL_CONSTANTS.C_MAX_MANIFOLDS DO
    L_Heating_Output_Active :=
        L_Heating_Output_Active
        OR GVL_HEATING_OUTPUT.DO_Manifold_Pumps[L_i]
        OR (GVL_HEATING_OUTPUT.AO_Manifold_Valves[L_i] > 0);
END_FOR;

L_Vent_Output_Active := GVL_VENT_OUTPUT.DO_Vent_Enable;
FOR L_i := 1 TO GVL_CONSTANTS.C_MAX_SUPPLY_FANS DO
    L_Vent_Output_Active :=
        L_Vent_Output_Active
        OR (GVL_VENT_OUTPUT.AO_Supply_Fans[L_i] > 0);
END_FOR;
FOR L_i := 1 TO GVL_CONSTANTS.C_MAX_EXHAUST_FANS DO
    L_Vent_Output_Active :=
        L_Vent_Output_Active
        OR (GVL_VENT_OUTPUT.AO_Exhaust_Fans[L_i] > 0);
END_FOR;

GVL_DOMAIN_EXECUTION_VALIDATION.Access_Stale_Output_Risk :=
    GVL_DOMAIN_EXECUTION_POLICY.Access_Idle_By_Design AND L_Access_Output_Active;

GVL_DOMAIN_EXECUTION_VALIDATION.Lighting_Stale_Output_Risk :=
    GVL_DOMAIN_EXECUTION_POLICY.Lighting_Idle_By_Design AND L_Lighting_Output_Active;

GVL_DOMAIN_EXECUTION_VALIDATION.Water_Stale_Output_Risk :=
    GVL_DOMAIN_EXECUTION_POLICY.Water_Idle_By_Design AND L_Water_Output_Active;

GVL_DOMAIN_EXECUTION_VALIDATION.Heating_Stale_Output_Risk :=
    GVL_DOMAIN_EXECUTION_POLICY.Heating_Idle_By_Design AND L_Heating_Output_Active;

GVL_DOMAIN_EXECUTION_VALIDATION.Vent_Stale_Output_Risk :=
    GVL_DOMAIN_EXECUTION_POLICY.Vent_Idle_By_Design AND L_Vent_Output_Active;

GVL_DOMAIN_EXECUTION_VALIDATION.Any_Stale_Output_Risk :=
    GVL_DOMAIN_EXECUTION_VALIDATION.Access_Stale_Output_Risk
    OR GVL_DOMAIN_EXECUTION_VALIDATION.Lighting_Stale_Output_Risk
    OR GVL_DOMAIN_EXECUTION_VALIDATION.Water_Stale_Output_Risk
    OR GVL_DOMAIN_EXECUTION_VALIDATION.Heating_Stale_Output_Risk
    OR GVL_DOMAIN_EXECUTION_VALIDATION.Vent_Stale_Output_Risk;

GVL_DOMAIN_EXECUTION_VALIDATION.Any_Policy_Mismatch :=
    GVL_DOMAIN_EXECUTION_VALIDATION.Any_Stale_Output_Risk;

IF GVL_DOMAIN_EXECUTION_VALIDATION.Any_Stale_Output_Risk THEN
    GVL_DOMAIN_EXECUTION_VALIDATION.G_Validation_Valid := FALSE;
    GVL_DOMAIN_EXECUTION_VALIDATION.Status_Code := 1;
    GVL_DOMAIN_EXECUTION_VALIDATION.Status_Text := 'Domain execution validation detected stale output risk';
ELSE
    GVL_DOMAIN_EXECUTION_VALIDATION.Status_Code := 0;
    GVL_DOMAIN_EXECUTION_VALIDATION.Status_Text := 'Domain execution validation nominal';
END_IF;

// >>> BULK_SYNC_ANCHOR: PRG_Domain_Execution_Validation <<<
END_PROGRAM

(* ---- PRG_DryRun_TestRig.st ---- *)
PROGRAM PRG_DryRun_TestRig
VAR
    fbDryRunHarness : FB_DryRun_Simulation_Harness;
    fbDryRunAssert  : FB_DryRun_Assertion_Map;

    L_DryRun_Enable : BOOL := FALSE;
    L_System_Time_MS : UDINT;

    L_Status_Line : STRING(120);
    L_Expected_Line : STRING(220);
END_VAR

// Local dry-run progression only.
// Not connected to production command/state paths yet.

fbDryRunHarness(
    VI_Enable := L_DryRun_Enable,
    VI_System_Time_MS := L_System_Time_MS,
    VO_Status_Msg => L_Status_Line
);

fbDryRunAssert(
    VI_Test_Step := fbDryRunHarness.VO_Test_Step,
    VO_Expected_Result => L_Expected_Line
);

// >>> BULK_SYNC_ANCHOR: PRG_DryRun_TestRig <<<

(* ---- PRG_Energy_Causality_Governor.st ---- *)
PROGRAM PRG_Energy_Causality_Governor
VAR
    L_Now_MS : UDINT;
    L_Energy_Valid : BOOL := TRUE;
    L_Error_Code : UDINT := 0;
    L_Error_Text : STRING(160) := '';
END_VAR

L_Now_MS := GVL_STATUS.G_System_Time_MS;
L_Energy_Valid := TRUE;
L_Error_Code := 0;
L_Error_Text := '';

// Fail-safe defaults.
GVL_ENERGY_CAUSALITY_FABRIC.Energy_Causality_Valid := FALSE;
GVL_ENERGY_CAUSALITY_FABRIC.Energy_Causality_Granted := FALSE;
GVL_ENERGY_CAUSALITY_FABRIC.Energy_Causality_Quarantine_Active := TRUE;

GVL_ENERGY_CAUSALITY_FABRIC.Hydraulic_Energy_State_Valid := FALSE;
GVL_ENERGY_CAUSALITY_FABRIC.Thermal_Energy_State_Valid := FALSE;
GVL_ENERGY_CAUSALITY_FABRIC.Electrical_Load_State_Valid := FALSE;
GVL_ENERGY_CAUSALITY_FABRIC.Motor_Energy_Envelope_Valid := FALSE;
GVL_ENERGY_CAUSALITY_FABRIC.Distributed_Load_Coherent := FALSE;

// Actuator semantic verification required.
IF NOT GVL_ACTUATOR_SEMANTIC_VERIFICATION.Actuator_Semantic_Verification_Granted THEN
    L_Energy_Valid := FALSE;
    L_Error_Code := 37000;
    L_Error_Text := 'Actuator semantic verification not granted';
END_IF;

// Energy divergence detectors.
IF GVL_ENERGY_CAUSALITY_FABRIC.DryRun_Energy_State_Detected THEN
    L_Energy_Valid := FALSE;
    L_Error_Code := 37001;
    L_Error_Text := 'Dry-run energy state detected';
END_IF;

IF GVL_ENERGY_CAUSALITY_FABRIC.Thermal_Extraction_Divergence_Detected THEN
    L_Energy_Valid := FALSE;
    L_Error_Code := 37002;
    L_Error_Text := 'Thermal extraction divergence detected';
END_IF;

IF GVL_ENERGY_CAUSALITY_FABRIC.Load_Synchronization_Spike_Detected THEN
    L_Energy_Valid := FALSE;
    L_Error_Code := 37003;
    L_Error_Text := 'Load synchronization spike detected';
END_IF;

IF GVL_ENERGY_CAUSALITY_FABRIC.Hydraulic_Energy_Starvation_Detected THEN
    L_Energy_Valid := FALSE;
    L_Error_Code := 37004;
    L_Error_Text := 'Hydraulic energy starvation detected';
END_IF;

IF GVL_ENERGY_CAUSALITY_FABRIC.Distributed_Transient_Overload_Detected THEN
    L_Energy_Valid := FALSE;
    L_Error_Code := 37005;
    L_Error_Text := 'Distributed transient overload detected';
END_IF;

IF GVL_ENERGY_CAUSALITY_FABRIC.Energy_Recovery_Instability_Detected THEN
    L_Energy_Valid := FALSE;
    L_Error_Code := 37006;
    L_Error_Text := 'Energy recovery instability detected';
END_IF;

// Stable energy envelope validation.
IF L_Energy_Valid
AND NOT GVL_ENERGY_CAUSALITY_FABRIC.Energy_Envelope_Stable THEN
    L_Energy_Valid := FALSE;
    L_Error_Code := 37010;
    L_Error_Text := 'Energy envelope unstable';
END_IF;

IF L_Energy_Valid
AND NOT GVL_ENERGY_CAUSALITY_FABRIC.Transient_Load_Stable THEN
    L_Energy_Valid := FALSE;
    L_Error_Code := 37011;
    L_Error_Text := 'Transient load stability invalid';
END_IF;

IF L_Energy_Valid
AND NOT GVL_ENERGY_CAUSALITY_FABRIC.Thermal_Accumulation_Stable THEN
    L_Energy_Valid := FALSE;
    L_Error_Code := 37012;
    L_Error_Text := 'Thermal accumulation unstable';
END_IF;

IF L_Energy_Valid
AND NOT GVL_ENERGY_CAUSALITY_FABRIC.Recovery_Energy_Coherent THEN
    L_Energy_Valid := FALSE;
    L_Error_Code := 37013;
    L_Error_Text := 'Recovery energy coherence invalid';
END_IF;

IF L_Energy_Valid THEN
    GVL_ENERGY_CAUSALITY_FABRIC.Energy_Causality_Valid := TRUE;
    GVL_ENERGY_CAUSALITY_FABRIC.Energy_Causality_Granted := TRUE;
    GVL_ENERGY_CAUSALITY_FABRIC.Energy_Causality_Quarantine_Active := FALSE;

    GVL_ENERGY_CAUSALITY_FABRIC.Hydraulic_Energy_State_Valid := TRUE;
    GVL_ENERGY_CAUSALITY_FABRIC.Thermal_Energy_State_Valid := TRUE;
    GVL_ENERGY_CAUSALITY_FABRIC.Electrical_Load_State_Valid := TRUE;
    GVL_ENERGY_CAUSALITY_FABRIC.Motor_Energy_Envelope_Valid := TRUE;
    GVL_ENERGY_CAUSALITY_FABRIC.Distributed_Load_Coherent := TRUE;

    GVL_ENERGY_CAUSALITY_FABRIC.Energy_Causality_Epoch :=
        GVL_ACTUATOR_SEMANTIC_VERIFICATION.Actuator_Verification_Epoch;

    GVL_ENERGY_CAUSALITY_FABRIC.Energy_Causality_Epoch_Coherent := TRUE;

    GVL_ENERGY_CAUSALITY_FABRIC.Energy_Causality_Last_Update_MS :=
        L_Now_MS;

    GVL_ENERGY_CAUSALITY_FABRIC.Energy_Causality_Lease_Expired := FALSE;

    GVL_ENERGY_CAUSALITY_FABRIC.Energy_Causality_Last_Error_Code := 0;
    GVL_ENERGY_CAUSALITY_FABRIC.Energy_Causality_Last_Error_Text := '';
ELSE
    GVL_ENERGY_CAUSALITY_FABRIC.Energy_Causality_Valid := FALSE;
    GVL_ENERGY_CAUSALITY_FABRIC.Energy_Causality_Granted := FALSE;
    GVL_ENERGY_CAUSALITY_FABRIC.Energy_Causality_Quarantine_Active := TRUE;

    GVL_ENERGY_CAUSALITY_FABRIC.Energy_Causality_Lease_Expired := TRUE;

    GVL_ENERGY_CAUSALITY_FABRIC.Energy_Causality_Last_Error_Code :=
        L_Error_Code;

    GVL_ENERGY_CAUSALITY_FABRIC.Energy_Causality_Last_Error_Text :=
        L_Error_Text;

    GVL_ENERGY_CAUSALITY_FABRIC.Energy_Causality_Invalidation_Count :=
        GVL_ENERGY_CAUSALITY_FABRIC.Energy_Causality_Invalidation_Count + 1;
END_IF;

END_PROGRAM
